   // UNICODE_TO_GBK[7258] := 16#5960;
   // UNICODE_TO_GBK[7259] := 16#B5EC;
   // UNICODE_TO_GBK[7260] := 16#5961;
   // UNICODE_TO_GBK[7261] := 16#8A53;
   // UNICODE_TO_GBK[7262] := 16#5962;
   // UNICODE_TO_GBK[7263] := 16#C9DD;
   // UNICODE_TO_GBK[7264] := 16#5963;
   // UNICODE_TO_GBK[7265] := 16#8A54;
   // UNICODE_TO_GBK[7266] := 16#5964;
   // UNICODE_TO_GBK[7267] := 16#8A55;
   // UNICODE_TO_GBK[7268] := 16#5965;
   // UNICODE_TO_GBK[7269] := 16#B0C2;
   // UNICODE_TO_GBK[7270] := 16#5966;
   // UNICODE_TO_GBK[7271] := 16#8A56;
   // UNICODE_TO_GBK[7272] := 16#5967;
   // UNICODE_TO_GBK[7273] := 16#8A57;
   // UNICODE_TO_GBK[7274] := 16#5968;
   // UNICODE_TO_GBK[7275] := 16#8A58;
   // UNICODE_TO_GBK[7276] := 16#5969;
   // UNICODE_TO_GBK[7277] := 16#8A59;
   // UNICODE_TO_GBK[7278] := 16#596A;
   // UNICODE_TO_GBK[7279] := 16#8A5A;
   // UNICODE_TO_GBK[7280] := 16#596B;
   // UNICODE_TO_GBK[7281] := 16#8A5B;
   // UNICODE_TO_GBK[7282] := 16#596C;
   // UNICODE_TO_GBK[7283] := 16#8A5C;
   // UNICODE_TO_GBK[7284] := 16#596D;
   // UNICODE_TO_GBK[7285] := 16#8A5D;
   // UNICODE_TO_GBK[7286] := 16#596E;
   // UNICODE_TO_GBK[7287] := 16#8A5E;
   // UNICODE_TO_GBK[7288] := 16#596F;
   // UNICODE_TO_GBK[7289] := 16#8A5F;
   // UNICODE_TO_GBK[7290] := 16#5970;
   // UNICODE_TO_GBK[7291] := 16#8A60;
   // UNICODE_TO_GBK[7292] := 16#5971;
   // UNICODE_TO_GBK[7293] := 16#8A61;
   // UNICODE_TO_GBK[7294] := 16#5972;
   // UNICODE_TO_GBK[7295] := 16#8A62;
   // UNICODE_TO_GBK[7296] := 16#5973;
   // UNICODE_TO_GBK[7297] := 16#C5AE;
   // UNICODE_TO_GBK[7298] := 16#5974;
   // UNICODE_TO_GBK[7299] := 16#C5AB;
   // UNICODE_TO_GBK[7300] := 16#5975;
   // UNICODE_TO_GBK[7301] := 16#8A63;
   // UNICODE_TO_GBK[7302] := 16#5976;
   // UNICODE_TO_GBK[7303] := 16#C4CC;
   // UNICODE_TO_GBK[7304] := 16#5977;
   // UNICODE_TO_GBK[7305] := 16#8A64;
   // UNICODE_TO_GBK[7306] := 16#5978;
   // UNICODE_TO_GBK[7307] := 16#BCE9;
   // UNICODE_TO_GBK[7308] := 16#5979;
   // UNICODE_TO_GBK[7309] := 16#CBFD;
   // UNICODE_TO_GBK[7310] := 16#597A;
   // UNICODE_TO_GBK[7311] := 16#8A65;
   // UNICODE_TO_GBK[7312] := 16#597B;
   // UNICODE_TO_GBK[7313] := 16#8A66;
   // UNICODE_TO_GBK[7314] := 16#597C;
   // UNICODE_TO_GBK[7315] := 16#8A67;
   // UNICODE_TO_GBK[7316] := 16#597D;
   // UNICODE_TO_GBK[7317] := 16#BAC3;
   // UNICODE_TO_GBK[7318] := 16#597E;
   // UNICODE_TO_GBK[7319] := 16#8A68;
   // UNICODE_TO_GBK[7320] := 16#597F;
   // UNICODE_TO_GBK[7321] := 16#8A69;
   // UNICODE_TO_GBK[7322] := 16#5980;
   // UNICODE_TO_GBK[7323] := 16#8A6A;
   // UNICODE_TO_GBK[7324] := 16#5981;
   // UNICODE_TO_GBK[7325] := 16#E5F9;
   // UNICODE_TO_GBK[7326] := 16#5982;
   // UNICODE_TO_GBK[7327] := 16#C8E7;
   // UNICODE_TO_GBK[7328] := 16#5983;
   // UNICODE_TO_GBK[7329] := 16#E5FA;
   // UNICODE_TO_GBK[7330] := 16#5984;
   // UNICODE_TO_GBK[7331] := 16#CDFD;
   // UNICODE_TO_GBK[7332] := 16#5985;
   // UNICODE_TO_GBK[7333] := 16#8A6B;
   // UNICODE_TO_GBK[7334] := 16#5986;
   // UNICODE_TO_GBK[7335] := 16#D7B1;
   // UNICODE_TO_GBK[7336] := 16#5987;
   // UNICODE_TO_GBK[7337] := 16#B8BE;
   // UNICODE_TO_GBK[7338] := 16#5988;
   // UNICODE_TO_GBK[7339] := 16#C2E8;
   // UNICODE_TO_GBK[7340] := 16#5989;
   // UNICODE_TO_GBK[7341] := 16#8A6C;
   // UNICODE_TO_GBK[7342] := 16#598A;
   // UNICODE_TO_GBK[7343] := 16#C8D1;
   // UNICODE_TO_GBK[7344] := 16#598B;
   // UNICODE_TO_GBK[7345] := 16#8A6D;
   // UNICODE_TO_GBK[7346] := 16#598C;
   // UNICODE_TO_GBK[7347] := 16#8A6E;
   // UNICODE_TO_GBK[7348] := 16#598D;
   // UNICODE_TO_GBK[7349] := 16#E5FB;
   // UNICODE_TO_GBK[7350] := 16#598E;
   // UNICODE_TO_GBK[7351] := 16#8A6F;
   // UNICODE_TO_GBK[7352] := 16#598F;
   // UNICODE_TO_GBK[7353] := 16#8A70;
   // UNICODE_TO_GBK[7354] := 16#5990;
   // UNICODE_TO_GBK[7355] := 16#8A71;
   // UNICODE_TO_GBK[7356] := 16#5991;
   // UNICODE_TO_GBK[7357] := 16#8A72;
   // UNICODE_TO_GBK[7358] := 16#5992;
   // UNICODE_TO_GBK[7359] := 16#B6CA;
   // UNICODE_TO_GBK[7360] := 16#5993;
   // UNICODE_TO_GBK[7361] := 16#BCCB;
   // UNICODE_TO_GBK[7362] := 16#5994;
   // UNICODE_TO_GBK[7363] := 16#8A73;
   // UNICODE_TO_GBK[7364] := 16#5995;
   // UNICODE_TO_GBK[7365] := 16#8A74;
   // UNICODE_TO_GBK[7366] := 16#5996;
   // UNICODE_TO_GBK[7367] := 16#D1FD;
   // UNICODE_TO_GBK[7368] := 16#5997;
   // UNICODE_TO_GBK[7369] := 16#E6A1;
   // UNICODE_TO_GBK[7370] := 16#5998;
   // UNICODE_TO_GBK[7371] := 16#8A75;
   // UNICODE_TO_GBK[7372] := 16#5999;
   // UNICODE_TO_GBK[7373] := 16#C3EE;
   // UNICODE_TO_GBK[7374] := 16#599A;
   // UNICODE_TO_GBK[7375] := 16#8A76;
   // UNICODE_TO_GBK[7376] := 16#599B;
   // UNICODE_TO_GBK[7377] := 16#8A77;
   // UNICODE_TO_GBK[7378] := 16#599C;
   // UNICODE_TO_GBK[7379] := 16#8A78;
   // UNICODE_TO_GBK[7380] := 16#599D;
   // UNICODE_TO_GBK[7381] := 16#8A79;
   // UNICODE_TO_GBK[7382] := 16#599E;
   // UNICODE_TO_GBK[7383] := 16#E6A4;
   // UNICODE_TO_GBK[7384] := 16#599F;
   // UNICODE_TO_GBK[7385] := 16#8A7A;
   // UNICODE_TO_GBK[7386] := 16#59A0;
   // UNICODE_TO_GBK[7387] := 16#8A7B;
   // UNICODE_TO_GBK[7388] := 16#59A1;
   // UNICODE_TO_GBK[7389] := 16#8A7C;
   // UNICODE_TO_GBK[7390] := 16#59A2;
   // UNICODE_TO_GBK[7391] := 16#8A7D;
   // UNICODE_TO_GBK[7392] := 16#59A3;
   // UNICODE_TO_GBK[7393] := 16#E5FE;
   // UNICODE_TO_GBK[7394] := 16#59A4;
   // UNICODE_TO_GBK[7395] := 16#E6A5;
   // UNICODE_TO_GBK[7396] := 16#59A5;
   // UNICODE_TO_GBK[7397] := 16#CDD7;
   // UNICODE_TO_GBK[7398] := 16#59A6;
   // UNICODE_TO_GBK[7399] := 16#8A7E;
   // UNICODE_TO_GBK[7400] := 16#59A7;
   // UNICODE_TO_GBK[7401] := 16#8A80;
   // UNICODE_TO_GBK[7402] := 16#59A8;
   // UNICODE_TO_GBK[7403] := 16#B7C1;
   // UNICODE_TO_GBK[7404] := 16#59A9;
   // UNICODE_TO_GBK[7405] := 16#E5FC;
   // UNICODE_TO_GBK[7406] := 16#59AA;
   // UNICODE_TO_GBK[7407] := 16#E5FD;
   // UNICODE_TO_GBK[7408] := 16#59AB;
   // UNICODE_TO_GBK[7409] := 16#E6A3;
   // UNICODE_TO_GBK[7410] := 16#59AC;
   // UNICODE_TO_GBK[7411] := 16#8A81;
   // UNICODE_TO_GBK[7412] := 16#59AD;
   // UNICODE_TO_GBK[7413] := 16#8A82;
   // UNICODE_TO_GBK[7414] := 16#59AE;
   // UNICODE_TO_GBK[7415] := 16#C4DD;
   // UNICODE_TO_GBK[7416] := 16#59AF;
   // UNICODE_TO_GBK[7417] := 16#E6A8;
   // UNICODE_TO_GBK[7418] := 16#59B0;
   // UNICODE_TO_GBK[7419] := 16#8A83;
   // UNICODE_TO_GBK[7420] := 16#59B1;
   // UNICODE_TO_GBK[7421] := 16#8A84;
   // UNICODE_TO_GBK[7422] := 16#59B2;
   // UNICODE_TO_GBK[7423] := 16#E6A7;
   // UNICODE_TO_GBK[7424] := 16#59B3;
   // UNICODE_TO_GBK[7425] := 16#8A85;
   // UNICODE_TO_GBK[7426] := 16#59B4;
   // UNICODE_TO_GBK[7427] := 16#8A86;
   // UNICODE_TO_GBK[7428] := 16#59B5;
   // UNICODE_TO_GBK[7429] := 16#8A87;
   // UNICODE_TO_GBK[7430] := 16#59B6;
   // UNICODE_TO_GBK[7431] := 16#8A88;
   // UNICODE_TO_GBK[7432] := 16#59B7;
   // UNICODE_TO_GBK[7433] := 16#8A89;
   // UNICODE_TO_GBK[7434] := 16#59B8;
   // UNICODE_TO_GBK[7435] := 16#8A8A;
   // UNICODE_TO_GBK[7436] := 16#59B9;
   // UNICODE_TO_GBK[7437] := 16#C3C3;
   // UNICODE_TO_GBK[7438] := 16#59BA;
   // UNICODE_TO_GBK[7439] := 16#8A8B;
   // UNICODE_TO_GBK[7440] := 16#59BB;
   // UNICODE_TO_GBK[7441] := 16#C6DE;
   // UNICODE_TO_GBK[7442] := 16#59BC;
   // UNICODE_TO_GBK[7443] := 16#8A8C;
   // UNICODE_TO_GBK[7444] := 16#59BD;
   // UNICODE_TO_GBK[7445] := 16#8A8D;
   // UNICODE_TO_GBK[7446] := 16#59BE;
   // UNICODE_TO_GBK[7447] := 16#E6AA;
   // UNICODE_TO_GBK[7448] := 16#59BF;
   // UNICODE_TO_GBK[7449] := 16#8A8E;
   // UNICODE_TO_GBK[7450] := 16#59C0;
   // UNICODE_TO_GBK[7451] := 16#8A8F;
   // UNICODE_TO_GBK[7452] := 16#59C1;
   // UNICODE_TO_GBK[7453] := 16#8A90;
   // UNICODE_TO_GBK[7454] := 16#59C2;
   // UNICODE_TO_GBK[7455] := 16#8A91;
   // UNICODE_TO_GBK[7456] := 16#59C3;
   // UNICODE_TO_GBK[7457] := 16#8A92;
   // UNICODE_TO_GBK[7458] := 16#59C4;
   // UNICODE_TO_GBK[7459] := 16#8A93;
   // UNICODE_TO_GBK[7460] := 16#59C5;
   // UNICODE_TO_GBK[7461] := 16#8A94;
   // UNICODE_TO_GBK[7462] := 16#59C6;
   // UNICODE_TO_GBK[7463] := 16#C4B7;
   // UNICODE_TO_GBK[7464] := 16#59C7;
   // UNICODE_TO_GBK[7465] := 16#8A95;
   // UNICODE_TO_GBK[7466] := 16#59C8;
   // UNICODE_TO_GBK[7467] := 16#8A96;
   // UNICODE_TO_GBK[7468] := 16#59C9;
   // UNICODE_TO_GBK[7469] := 16#8A97;
   // UNICODE_TO_GBK[7470] := 16#59CA;
   // UNICODE_TO_GBK[7471] := 16#E6A2;
   // UNICODE_TO_GBK[7472] := 16#59CB;
   // UNICODE_TO_GBK[7473] := 16#CABC;
   // UNICODE_TO_GBK[7474] := 16#59CC;
   // UNICODE_TO_GBK[7475] := 16#8A98;
   // UNICODE_TO_GBK[7476] := 16#59CD;
   // UNICODE_TO_GBK[7477] := 16#8A99;
   // UNICODE_TO_GBK[7478] := 16#59CE;
   // UNICODE_TO_GBK[7479] := 16#8A9A;
   // UNICODE_TO_GBK[7480] := 16#59CF;
   // UNICODE_TO_GBK[7481] := 16#8A9B;
   // UNICODE_TO_GBK[7482] := 16#59D0;
   // UNICODE_TO_GBK[7483] := 16#BDE3;
   // UNICODE_TO_GBK[7484] := 16#59D1;
   // UNICODE_TO_GBK[7485] := 16#B9C3;
   // UNICODE_TO_GBK[7486] := 16#59D2;
   // UNICODE_TO_GBK[7487] := 16#E6A6;
   // UNICODE_TO_GBK[7488] := 16#59D3;
   // UNICODE_TO_GBK[7489] := 16#D0D5;
   // UNICODE_TO_GBK[7490] := 16#59D4;
   // UNICODE_TO_GBK[7491] := 16#CEAF;
   // UNICODE_TO_GBK[7492] := 16#59D5;
   // UNICODE_TO_GBK[7493] := 16#8A9C;
   // UNICODE_TO_GBK[7494] := 16#59D6;
   // UNICODE_TO_GBK[7495] := 16#8A9D;
   // UNICODE_TO_GBK[7496] := 16#59D7;
   // UNICODE_TO_GBK[7497] := 16#E6A9;
   // UNICODE_TO_GBK[7498] := 16#59D8;
   // UNICODE_TO_GBK[7499] := 16#E6B0;
   // UNICODE_TO_GBK[7500] := 16#59D9;
   // UNICODE_TO_GBK[7501] := 16#8A9E;
   // UNICODE_TO_GBK[7502] := 16#59DA;
   // UNICODE_TO_GBK[7503] := 16#D2A6;
   // UNICODE_TO_GBK[7504] := 16#59DB;
   // UNICODE_TO_GBK[7505] := 16#8A9F;
   // UNICODE_TO_GBK[7506] := 16#59DC;
   // UNICODE_TO_GBK[7507] := 16#BDAA;
   // UNICODE_TO_GBK[7508] := 16#59DD;
   // UNICODE_TO_GBK[7509] := 16#E6AD;
   // UNICODE_TO_GBK[7510] := 16#59DE;
   // UNICODE_TO_GBK[7511] := 16#8AA0;
   // UNICODE_TO_GBK[7512] := 16#59DF;
   // UNICODE_TO_GBK[7513] := 16#8AA1;
   // UNICODE_TO_GBK[7514] := 16#59E0;
   // UNICODE_TO_GBK[7515] := 16#8AA2;
   // UNICODE_TO_GBK[7516] := 16#59E1;
   // UNICODE_TO_GBK[7517] := 16#8AA3;
   // UNICODE_TO_GBK[7518] := 16#59E2;
   // UNICODE_TO_GBK[7519] := 16#8AA4;
   // UNICODE_TO_GBK[7520] := 16#59E3;
   // UNICODE_TO_GBK[7521] := 16#E6AF;
   // UNICODE_TO_GBK[7522] := 16#59E4;
   // UNICODE_TO_GBK[7523] := 16#8AA5;
   // UNICODE_TO_GBK[7524] := 16#59E5;
   // UNICODE_TO_GBK[7525] := 16#C0D1;
   // UNICODE_TO_GBK[7526] := 16#59E6;
   // UNICODE_TO_GBK[7527] := 16#8AA6;
   // UNICODE_TO_GBK[7528] := 16#59E7;
   // UNICODE_TO_GBK[7529] := 16#8AA7;
   // UNICODE_TO_GBK[7530] := 16#59E8;
   // UNICODE_TO_GBK[7531] := 16#D2CC;
   // UNICODE_TO_GBK[7532] := 16#59E9;
   // UNICODE_TO_GBK[7533] := 16#8AA8;
   // UNICODE_TO_GBK[7534] := 16#59EA;
   // UNICODE_TO_GBK[7535] := 16#8AA9;
   // UNICODE_TO_GBK[7536] := 16#59EB;
   // UNICODE_TO_GBK[7537] := 16#8AAA;
   // UNICODE_TO_GBK[7538] := 16#59EC;
   // UNICODE_TO_GBK[7539] := 16#BCA7;
   // UNICODE_TO_GBK[7540] := 16#59ED;
   // UNICODE_TO_GBK[7541] := 16#8AAB;
   // UNICODE_TO_GBK[7542] := 16#59EE;
   // UNICODE_TO_GBK[7543] := 16#8AAC;
   // UNICODE_TO_GBK[7544] := 16#59EF;
   // UNICODE_TO_GBK[7545] := 16#8AAD;
   // UNICODE_TO_GBK[7546] := 16#59F0;
   // UNICODE_TO_GBK[7547] := 16#8AAE;
   // UNICODE_TO_GBK[7548] := 16#59F1;
   // UNICODE_TO_GBK[7549] := 16#8AAF;
   // UNICODE_TO_GBK[7550] := 16#59F2;
   // UNICODE_TO_GBK[7551] := 16#8AB0;
   // UNICODE_TO_GBK[7552] := 16#59F3;
   // UNICODE_TO_GBK[7553] := 16#8AB1;
   // UNICODE_TO_GBK[7554] := 16#59F4;
   // UNICODE_TO_GBK[7555] := 16#8AB2;
   // UNICODE_TO_GBK[7556] := 16#59F5;
   // UNICODE_TO_GBK[7557] := 16#8AB3;
   // UNICODE_TO_GBK[7558] := 16#59F6;
   // UNICODE_TO_GBK[7559] := 16#8AB4;
   // UNICODE_TO_GBK[7560] := 16#59F7;
   // UNICODE_TO_GBK[7561] := 16#8AB5;
   // UNICODE_TO_GBK[7562] := 16#59F8;
   // UNICODE_TO_GBK[7563] := 16#8AB6;
   // UNICODE_TO_GBK[7564] := 16#59F9;
   // UNICODE_TO_GBK[7565] := 16#E6B1;
   // UNICODE_TO_GBK[7566] := 16#59FA;
   // UNICODE_TO_GBK[7567] := 16#8AB7;
   // UNICODE_TO_GBK[7568] := 16#59FB;
   // UNICODE_TO_GBK[7569] := 16#D2F6;
   // UNICODE_TO_GBK[7570] := 16#59FC;
   // UNICODE_TO_GBK[7571] := 16#8AB8;
   // UNICODE_TO_GBK[7572] := 16#59FD;
   // UNICODE_TO_GBK[7573] := 16#8AB9;
   // UNICODE_TO_GBK[7574] := 16#59FE;
   // UNICODE_TO_GBK[7575] := 16#8ABA;
   // UNICODE_TO_GBK[7576] := 16#59FF;
   // UNICODE_TO_GBK[7577] := 16#D7CB;
   // UNICODE_TO_GBK[7578] := 16#5A00;
   // UNICODE_TO_GBK[7579] := 16#8ABB;
   // UNICODE_TO_GBK[7580] := 16#5A01;
   // UNICODE_TO_GBK[7581] := 16#CDFE;
   // UNICODE_TO_GBK[7582] := 16#5A02;
   // UNICODE_TO_GBK[7583] := 16#8ABC;
   // UNICODE_TO_GBK[7584] := 16#5A03;
   // UNICODE_TO_GBK[7585] := 16#CDDE;
   // UNICODE_TO_GBK[7586] := 16#5A04;
   // UNICODE_TO_GBK[7587] := 16#C2A6;
   // UNICODE_TO_GBK[7588] := 16#5A05;
   // UNICODE_TO_GBK[7589] := 16#E6AB;
   // UNICODE_TO_GBK[7590] := 16#5A06;
   // UNICODE_TO_GBK[7591] := 16#E6AC;
   // UNICODE_TO_GBK[7592] := 16#5A07;
   // UNICODE_TO_GBK[7593] := 16#BDBF;
   // UNICODE_TO_GBK[7594] := 16#5A08;
   // UNICODE_TO_GBK[7595] := 16#E6AE;
   // UNICODE_TO_GBK[7596] := 16#5A09;
   // UNICODE_TO_GBK[7597] := 16#E6B3;
   // UNICODE_TO_GBK[7598] := 16#5A0A;
   // UNICODE_TO_GBK[7599] := 16#8ABD;
   // UNICODE_TO_GBK[7600] := 16#5A0B;
   // UNICODE_TO_GBK[7601] := 16#8ABE;
   // UNICODE_TO_GBK[7602] := 16#5A0C;
   // UNICODE_TO_GBK[7603] := 16#E6B2;
   // UNICODE_TO_GBK[7604] := 16#5A0D;
   // UNICODE_TO_GBK[7605] := 16#8ABF;
   // UNICODE_TO_GBK[7606] := 16#5A0E;
   // UNICODE_TO_GBK[7607] := 16#8AC0;
   // UNICODE_TO_GBK[7608] := 16#5A0F;
   // UNICODE_TO_GBK[7609] := 16#8AC1;
   // UNICODE_TO_GBK[7610] := 16#5A10;
   // UNICODE_TO_GBK[7611] := 16#8AC2;
   // UNICODE_TO_GBK[7612] := 16#5A11;
   // UNICODE_TO_GBK[7613] := 16#E6B6;
   // UNICODE_TO_GBK[7614] := 16#5A12;
   // UNICODE_TO_GBK[7615] := 16#8AC3;
   // UNICODE_TO_GBK[7616] := 16#5A13;
   // UNICODE_TO_GBK[7617] := 16#E6B8;
   // UNICODE_TO_GBK[7618] := 16#5A14;
   // UNICODE_TO_GBK[7619] := 16#8AC4;
   // UNICODE_TO_GBK[7620] := 16#5A15;
   // UNICODE_TO_GBK[7621] := 16#8AC5;
   // UNICODE_TO_GBK[7622] := 16#5A16;
   // UNICODE_TO_GBK[7623] := 16#8AC6;
   // UNICODE_TO_GBK[7624] := 16#5A17;
   // UNICODE_TO_GBK[7625] := 16#8AC7;
   // UNICODE_TO_GBK[7626] := 16#5A18;
   // UNICODE_TO_GBK[7627] := 16#C4EF;
   // UNICODE_TO_GBK[7628] := 16#5A19;
   // UNICODE_TO_GBK[7629] := 16#8AC8;
   // UNICODE_TO_GBK[7630] := 16#5A1A;
   // UNICODE_TO_GBK[7631] := 16#8AC9;
   // UNICODE_TO_GBK[7632] := 16#5A1B;
   // UNICODE_TO_GBK[7633] := 16#8ACA;
   // UNICODE_TO_GBK[7634] := 16#5A1C;
   // UNICODE_TO_GBK[7635] := 16#C4C8;
   // UNICODE_TO_GBK[7636] := 16#5A1D;
   // UNICODE_TO_GBK[7637] := 16#8ACB;
   // UNICODE_TO_GBK[7638] := 16#5A1E;
   // UNICODE_TO_GBK[7639] := 16#8ACC;
   // UNICODE_TO_GBK[7640] := 16#5A1F;
   // UNICODE_TO_GBK[7641] := 16#BEEA;
   // UNICODE_TO_GBK[7642] := 16#5A20;
   // UNICODE_TO_GBK[7643] := 16#C9EF;
   // UNICODE_TO_GBK[7644] := 16#5A21;
   // UNICODE_TO_GBK[7645] := 16#8ACD;
   // UNICODE_TO_GBK[7646] := 16#5A22;
   // UNICODE_TO_GBK[7647] := 16#8ACE;
   // UNICODE_TO_GBK[7648] := 16#5A23;
   // UNICODE_TO_GBK[7649] := 16#E6B7;
   // UNICODE_TO_GBK[7650] := 16#5A24;
   // UNICODE_TO_GBK[7651] := 16#8ACF;
   // UNICODE_TO_GBK[7652] := 16#5A25;
   // UNICODE_TO_GBK[7653] := 16#B6F0;
   // UNICODE_TO_GBK[7654] := 16#5A26;
   // UNICODE_TO_GBK[7655] := 16#8AD0;
   // UNICODE_TO_GBK[7656] := 16#5A27;
   // UNICODE_TO_GBK[7657] := 16#8AD1;
   // UNICODE_TO_GBK[7658] := 16#5A28;
   // UNICODE_TO_GBK[7659] := 16#8AD2;
   // UNICODE_TO_GBK[7660] := 16#5A29;
   // UNICODE_TO_GBK[7661] := 16#C3E4;
   // UNICODE_TO_GBK[7662] := 16#5A2A;
   // UNICODE_TO_GBK[7663] := 16#8AD3;
   // UNICODE_TO_GBK[7664] := 16#5A2B;
   // UNICODE_TO_GBK[7665] := 16#8AD4;
   // UNICODE_TO_GBK[7666] := 16#5A2C;
   // UNICODE_TO_GBK[7667] := 16#8AD5;
   // UNICODE_TO_GBK[7668] := 16#5A2D;
   // UNICODE_TO_GBK[7669] := 16#8AD6;
   // UNICODE_TO_GBK[7670] := 16#5A2E;
   // UNICODE_TO_GBK[7671] := 16#8AD7;
   // UNICODE_TO_GBK[7672] := 16#5A2F;
   // UNICODE_TO_GBK[7673] := 16#8AD8;
   // UNICODE_TO_GBK[7674] := 16#5A30;
   // UNICODE_TO_GBK[7675] := 16#8AD9;
   // UNICODE_TO_GBK[7676] := 16#5A31;
   // UNICODE_TO_GBK[7677] := 16#D3E9;
   // UNICODE_TO_GBK[7678] := 16#5A32;
   // UNICODE_TO_GBK[7679] := 16#E6B4;
   // UNICODE_TO_GBK[7680] := 16#5A33;
   // UNICODE_TO_GBK[7681] := 16#8ADA;
   // UNICODE_TO_GBK[7682] := 16#5A34;
   // UNICODE_TO_GBK[7683] := 16#E6B5;
   // UNICODE_TO_GBK[7684] := 16#5A35;
   // UNICODE_TO_GBK[7685] := 16#8ADB;
   // UNICODE_TO_GBK[7686] := 16#5A36;
   // UNICODE_TO_GBK[7687] := 16#C8A2;
   // UNICODE_TO_GBK[7688] := 16#5A37;
   // UNICODE_TO_GBK[7689] := 16#8ADC;
   // UNICODE_TO_GBK[7690] := 16#5A38;
   // UNICODE_TO_GBK[7691] := 16#8ADD;
   // UNICODE_TO_GBK[7692] := 16#5A39;
   // UNICODE_TO_GBK[7693] := 16#8ADE;
   // UNICODE_TO_GBK[7694] := 16#5A3A;
   // UNICODE_TO_GBK[7695] := 16#8ADF;
   // UNICODE_TO_GBK[7696] := 16#5A3B;
   // UNICODE_TO_GBK[7697] := 16#8AE0;
   // UNICODE_TO_GBK[7698] := 16#5A3C;
   // UNICODE_TO_GBK[7699] := 16#E6BD;
   // UNICODE_TO_GBK[7700] := 16#5A3D;
   // UNICODE_TO_GBK[7701] := 16#8AE1;
   // UNICODE_TO_GBK[7702] := 16#5A3E;
   // UNICODE_TO_GBK[7703] := 16#8AE2;
   // UNICODE_TO_GBK[7704] := 16#5A3F;
   // UNICODE_TO_GBK[7705] := 16#8AE3;
   // UNICODE_TO_GBK[7706] := 16#5A40;
   // UNICODE_TO_GBK[7707] := 16#E6B9;
   // UNICODE_TO_GBK[7708] := 16#5A41;
   // UNICODE_TO_GBK[7709] := 16#8AE4;
   // UNICODE_TO_GBK[7710] := 16#5A42;
   // UNICODE_TO_GBK[7711] := 16#8AE5;
   // UNICODE_TO_GBK[7712] := 16#5A43;
   // UNICODE_TO_GBK[7713] := 16#8AE6;
   // UNICODE_TO_GBK[7714] := 16#5A44;
   // UNICODE_TO_GBK[7715] := 16#8AE7;
   // UNICODE_TO_GBK[7716] := 16#5A45;
   // UNICODE_TO_GBK[7717] := 16#8AE8;
   // UNICODE_TO_GBK[7718] := 16#5A46;
   // UNICODE_TO_GBK[7719] := 16#C6C5;
   // UNICODE_TO_GBK[7720] := 16#5A47;
   // UNICODE_TO_GBK[7721] := 16#8AE9;
   // UNICODE_TO_GBK[7722] := 16#5A48;
   // UNICODE_TO_GBK[7723] := 16#8AEA;
   // UNICODE_TO_GBK[7724] := 16#5A49;
   // UNICODE_TO_GBK[7725] := 16#CDF1;
   // UNICODE_TO_GBK[7726] := 16#5A4A;
   // UNICODE_TO_GBK[7727] := 16#E6BB;
   // UNICODE_TO_GBK[7728] := 16#5A4B;
   // UNICODE_TO_GBK[7729] := 16#8AEB;
   // UNICODE_TO_GBK[7730] := 16#5A4C;
   // UNICODE_TO_GBK[7731] := 16#8AEC;
   // UNICODE_TO_GBK[7732] := 16#5A4D;
   // UNICODE_TO_GBK[7733] := 16#8AED;
   // UNICODE_TO_GBK[7734] := 16#5A4E;
   // UNICODE_TO_GBK[7735] := 16#8AEE;
   // UNICODE_TO_GBK[7736] := 16#5A4F;
   // UNICODE_TO_GBK[7737] := 16#8AEF;
   // UNICODE_TO_GBK[7738] := 16#5A50;
   // UNICODE_TO_GBK[7739] := 16#8AF0;
   // UNICODE_TO_GBK[7740] := 16#5A51;
   // UNICODE_TO_GBK[7741] := 16#8AF1;
   // UNICODE_TO_GBK[7742] := 16#5A52;
   // UNICODE_TO_GBK[7743] := 16#8AF2;
   // UNICODE_TO_GBK[7744] := 16#5A53;
   // UNICODE_TO_GBK[7745] := 16#8AF3;
   // UNICODE_TO_GBK[7746] := 16#5A54;
   // UNICODE_TO_GBK[7747] := 16#8AF4;
   // UNICODE_TO_GBK[7748] := 16#5A55;
   // UNICODE_TO_GBK[7749] := 16#E6BC;
   // UNICODE_TO_GBK[7750] := 16#5A56;
   // UNICODE_TO_GBK[7751] := 16#8AF5;
   // UNICODE_TO_GBK[7752] := 16#5A57;
   // UNICODE_TO_GBK[7753] := 16#8AF6;
   // UNICODE_TO_GBK[7754] := 16#5A58;
   // UNICODE_TO_GBK[7755] := 16#8AF7;
   // UNICODE_TO_GBK[7756] := 16#5A59;
   // UNICODE_TO_GBK[7757] := 16#8AF8;
   // UNICODE_TO_GBK[7758] := 16#5A5A;
   // UNICODE_TO_GBK[7759] := 16#BBE9;
   // UNICODE_TO_GBK[7760] := 16#5A5B;
   // UNICODE_TO_GBK[7761] := 16#8AF9;
   // UNICODE_TO_GBK[7762] := 16#5A5C;
   // UNICODE_TO_GBK[7763] := 16#8AFA;
   // UNICODE_TO_GBK[7764] := 16#5A5D;
   // UNICODE_TO_GBK[7765] := 16#8AFB;
   // UNICODE_TO_GBK[7766] := 16#5A5E;
   // UNICODE_TO_GBK[7767] := 16#8AFC;
   // UNICODE_TO_GBK[7768] := 16#5A5F;
   // UNICODE_TO_GBK[7769] := 16#8AFD;
   // UNICODE_TO_GBK[7770] := 16#5A60;
   // UNICODE_TO_GBK[7771] := 16#8AFE;
   // UNICODE_TO_GBK[7772] := 16#5A61;
   // UNICODE_TO_GBK[7773] := 16#8B40;
   // UNICODE_TO_GBK[7774] := 16#5A62;
   // UNICODE_TO_GBK[7775] := 16#E6BE;
   // UNICODE_TO_GBK[7776] := 16#5A63;
   // UNICODE_TO_GBK[7777] := 16#8B41;
   // UNICODE_TO_GBK[7778] := 16#5A64;
   // UNICODE_TO_GBK[7779] := 16#8B42;
   // UNICODE_TO_GBK[7780] := 16#5A65;
   // UNICODE_TO_GBK[7781] := 16#8B43;
   // UNICODE_TO_GBK[7782] := 16#5A66;
   // UNICODE_TO_GBK[7783] := 16#8B44;
   // UNICODE_TO_GBK[7784] := 16#5A67;
   // UNICODE_TO_GBK[7785] := 16#E6BA;
   // UNICODE_TO_GBK[7786] := 16#5A68;
   // UNICODE_TO_GBK[7787] := 16#8B45;
   // UNICODE_TO_GBK[7788] := 16#5A69;
   // UNICODE_TO_GBK[7789] := 16#8B46;
   // UNICODE_TO_GBK[7790] := 16#5A6A;
   // UNICODE_TO_GBK[7791] := 16#C0B7;
   // UNICODE_TO_GBK[7792] := 16#5A6B;
   // UNICODE_TO_GBK[7793] := 16#8B47;
   // UNICODE_TO_GBK[7794] := 16#5A6C;
   // UNICODE_TO_GBK[7795] := 16#8B48;
   // UNICODE_TO_GBK[7796] := 16#5A6D;
   // UNICODE_TO_GBK[7797] := 16#8B49;
   // UNICODE_TO_GBK[7798] := 16#5A6E;
   // UNICODE_TO_GBK[7799] := 16#8B4A;
   // UNICODE_TO_GBK[7800] := 16#5A6F;
   // UNICODE_TO_GBK[7801] := 16#8B4B;
   // UNICODE_TO_GBK[7802] := 16#5A70;
   // UNICODE_TO_GBK[7803] := 16#8B4C;
   // UNICODE_TO_GBK[7804] := 16#5A71;
   // UNICODE_TO_GBK[7805] := 16#8B4D;
   // UNICODE_TO_GBK[7806] := 16#5A72;
   // UNICODE_TO_GBK[7807] := 16#8B4E;
   // UNICODE_TO_GBK[7808] := 16#5A73;
   // UNICODE_TO_GBK[7809] := 16#8B4F;
   // UNICODE_TO_GBK[7810] := 16#5A74;
   // UNICODE_TO_GBK[7811] := 16#D3A4;
   // UNICODE_TO_GBK[7812] := 16#5A75;
   // UNICODE_TO_GBK[7813] := 16#E6BF;
   // UNICODE_TO_GBK[7814] := 16#5A76;
   // UNICODE_TO_GBK[7815] := 16#C9F4;
   // UNICODE_TO_GBK[7816] := 16#5A77;
   // UNICODE_TO_GBK[7817] := 16#E6C3;
   // UNICODE_TO_GBK[7818] := 16#5A78;
   // UNICODE_TO_GBK[7819] := 16#8B50;
   // UNICODE_TO_GBK[7820] := 16#5A79;
   // UNICODE_TO_GBK[7821] := 16#8B51;
   // UNICODE_TO_GBK[7822] := 16#5A7A;
   // UNICODE_TO_GBK[7823] := 16#E6C4;
   // UNICODE_TO_GBK[7824] := 16#5A7B;
   // UNICODE_TO_GBK[7825] := 16#8B52;
   // UNICODE_TO_GBK[7826] := 16#5A7C;
   // UNICODE_TO_GBK[7827] := 16#8B53;
   // UNICODE_TO_GBK[7828] := 16#5A7D;
   // UNICODE_TO_GBK[7829] := 16#8B54;
   // UNICODE_TO_GBK[7830] := 16#5A7E;
   // UNICODE_TO_GBK[7831] := 16#8B55;
   // UNICODE_TO_GBK[7832] := 16#5A7F;
   // UNICODE_TO_GBK[7833] := 16#D0F6;
   // UNICODE_TO_GBK[7834] := 16#5A80;
   // UNICODE_TO_GBK[7835] := 16#8B56;
   // UNICODE_TO_GBK[7836] := 16#5A81;
   // UNICODE_TO_GBK[7837] := 16#8B57;
   // UNICODE_TO_GBK[7838] := 16#5A82;
   // UNICODE_TO_GBK[7839] := 16#8B58;
   // UNICODE_TO_GBK[7840] := 16#5A83;
   // UNICODE_TO_GBK[7841] := 16#8B59;
   // UNICODE_TO_GBK[7842] := 16#5A84;
   // UNICODE_TO_GBK[7843] := 16#8B5A;
   // UNICODE_TO_GBK[7844] := 16#5A85;
   // UNICODE_TO_GBK[7845] := 16#8B5B;
   // UNICODE_TO_GBK[7846] := 16#5A86;
   // UNICODE_TO_GBK[7847] := 16#8B5C;
   // UNICODE_TO_GBK[7848] := 16#5A87;
   // UNICODE_TO_GBK[7849] := 16#8B5D;
   // UNICODE_TO_GBK[7850] := 16#5A88;
   // UNICODE_TO_GBK[7851] := 16#8B5E;
   // UNICODE_TO_GBK[7852] := 16#5A89;
   // UNICODE_TO_GBK[7853] := 16#8B5F;
   // UNICODE_TO_GBK[7854] := 16#5A8A;
   // UNICODE_TO_GBK[7855] := 16#8B60;
   // UNICODE_TO_GBK[7856] := 16#5A8B;
   // UNICODE_TO_GBK[7857] := 16#8B61;
   // UNICODE_TO_GBK[7858] := 16#5A8C;
   // UNICODE_TO_GBK[7859] := 16#8B62;
   // UNICODE_TO_GBK[7860] := 16#5A8D;
   // UNICODE_TO_GBK[7861] := 16#8B63;
   // UNICODE_TO_GBK[7862] := 16#5A8E;
   // UNICODE_TO_GBK[7863] := 16#8B64;
   // UNICODE_TO_GBK[7864] := 16#5A8F;
   // UNICODE_TO_GBK[7865] := 16#8B65;
   // UNICODE_TO_GBK[7866] := 16#5A90;
   // UNICODE_TO_GBK[7867] := 16#8B66;
   // UNICODE_TO_GBK[7868] := 16#5A91;
   // UNICODE_TO_GBK[7869] := 16#8B67;
   // UNICODE_TO_GBK[7870] := 16#5A92;
   // UNICODE_TO_GBK[7871] := 16#C3BD;
   // UNICODE_TO_GBK[7872] := 16#5A93;
   // UNICODE_TO_GBK[7873] := 16#8B68;
   // UNICODE_TO_GBK[7874] := 16#5A94;
   // UNICODE_TO_GBK[7875] := 16#8B69;
   // UNICODE_TO_GBK[7876] := 16#5A95;
   // UNICODE_TO_GBK[7877] := 16#8B6A;
   // UNICODE_TO_GBK[7878] := 16#5A96;
   // UNICODE_TO_GBK[7879] := 16#8B6B;
   // UNICODE_TO_GBK[7880] := 16#5A97;
   // UNICODE_TO_GBK[7881] := 16#8B6C;
   // UNICODE_TO_GBK[7882] := 16#5A98;
   // UNICODE_TO_GBK[7883] := 16#8B6D;
   // UNICODE_TO_GBK[7884] := 16#5A99;
   // UNICODE_TO_GBK[7885] := 16#8B6E;
   // UNICODE_TO_GBK[7886] := 16#5A9A;
   // UNICODE_TO_GBK[7887] := 16#C3C4;
   // UNICODE_TO_GBK[7888] := 16#5A9B;
   // UNICODE_TO_GBK[7889] := 16#E6C2;
   // UNICODE_TO_GBK[7890] := 16#5A9C;
   // UNICODE_TO_GBK[7891] := 16#8B6F;
   // UNICODE_TO_GBK[7892] := 16#5A9D;
   // UNICODE_TO_GBK[7893] := 16#8B70;
   // UNICODE_TO_GBK[7894] := 16#5A9E;
   // UNICODE_TO_GBK[7895] := 16#8B71;
   // UNICODE_TO_GBK[7896] := 16#5A9F;
   // UNICODE_TO_GBK[7897] := 16#8B72;
   // UNICODE_TO_GBK[7898] := 16#5AA0;
   // UNICODE_TO_GBK[7899] := 16#8B73;
   // UNICODE_TO_GBK[7900] := 16#5AA1;
   // UNICODE_TO_GBK[7901] := 16#8B74;
   // UNICODE_TO_GBK[7902] := 16#5AA2;
   // UNICODE_TO_GBK[7903] := 16#8B75;
   // UNICODE_TO_GBK[7904] := 16#5AA3;
   // UNICODE_TO_GBK[7905] := 16#8B76;
   // UNICODE_TO_GBK[7906] := 16#5AA4;
   // UNICODE_TO_GBK[7907] := 16#8B77;
   // UNICODE_TO_GBK[7908] := 16#5AA5;
   // UNICODE_TO_GBK[7909] := 16#8B78;
   // UNICODE_TO_GBK[7910] := 16#5AA6;
   // UNICODE_TO_GBK[7911] := 16#8B79;
   // UNICODE_TO_GBK[7912] := 16#5AA7;
   // UNICODE_TO_GBK[7913] := 16#8B7A;
   // UNICODE_TO_GBK[7914] := 16#5AA8;
   // UNICODE_TO_GBK[7915] := 16#8B7B;
   // UNICODE_TO_GBK[7916] := 16#5AA9;
   // UNICODE_TO_GBK[7917] := 16#8B7C;
   // UNICODE_TO_GBK[7918] := 16#5AAA;
   // UNICODE_TO_GBK[7919] := 16#E6C1;
   // UNICODE_TO_GBK[7920] := 16#5AAB;
   // UNICODE_TO_GBK[7921] := 16#8B7D;
   // UNICODE_TO_GBK[7922] := 16#5AAC;
   // UNICODE_TO_GBK[7923] := 16#8B7E;
   // UNICODE_TO_GBK[7924] := 16#5AAD;
   // UNICODE_TO_GBK[7925] := 16#8B80;
   // UNICODE_TO_GBK[7926] := 16#5AAE;
   // UNICODE_TO_GBK[7927] := 16#8B81;
   // UNICODE_TO_GBK[7928] := 16#5AAF;
   // UNICODE_TO_GBK[7929] := 16#8B82;
   // UNICODE_TO_GBK[7930] := 16#5AB0;
   // UNICODE_TO_GBK[7931] := 16#8B83;
   // UNICODE_TO_GBK[7932] := 16#5AB1;
   // UNICODE_TO_GBK[7933] := 16#8B84;
   // UNICODE_TO_GBK[7934] := 16#5AB2;
   // UNICODE_TO_GBK[7935] := 16#E6C7;
   // UNICODE_TO_GBK[7936] := 16#5AB3;
   // UNICODE_TO_GBK[7937] := 16#CFB1;
   // UNICODE_TO_GBK[7938] := 16#5AB4;
   // UNICODE_TO_GBK[7939] := 16#8B85;
   // UNICODE_TO_GBK[7940] := 16#5AB5;
   // UNICODE_TO_GBK[7941] := 16#EBF4;
   // UNICODE_TO_GBK[7942] := 16#5AB6;
   // UNICODE_TO_GBK[7943] := 16#8B86;
   // UNICODE_TO_GBK[7944] := 16#5AB7;
   // UNICODE_TO_GBK[7945] := 16#8B87;
   // UNICODE_TO_GBK[7946] := 16#5AB8;
   // UNICODE_TO_GBK[7947] := 16#E6CA;
   // UNICODE_TO_GBK[7948] := 16#5AB9;
   // UNICODE_TO_GBK[7949] := 16#8B88;
   // UNICODE_TO_GBK[7950] := 16#5ABA;
   // UNICODE_TO_GBK[7951] := 16#8B89;
   // UNICODE_TO_GBK[7952] := 16#5ABB;
   // UNICODE_TO_GBK[7953] := 16#8B8A;
   // UNICODE_TO_GBK[7954] := 16#5ABC;
   // UNICODE_TO_GBK[7955] := 16#8B8B;
   // UNICODE_TO_GBK[7956] := 16#5ABD;
   // UNICODE_TO_GBK[7957] := 16#8B8C;
   // UNICODE_TO_GBK[7958] := 16#5ABE;
   // UNICODE_TO_GBK[7959] := 16#E6C5;
   // UNICODE_TO_GBK[7960] := 16#5ABF;
   // UNICODE_TO_GBK[7961] := 16#8B8D;
   // UNICODE_TO_GBK[7962] := 16#5AC0;
   // UNICODE_TO_GBK[7963] := 16#8B8E;
   // UNICODE_TO_GBK[7964] := 16#5AC1;
   // UNICODE_TO_GBK[7965] := 16#BCDE;
   // UNICODE_TO_GBK[7966] := 16#5AC2;
   // UNICODE_TO_GBK[7967] := 16#C9A9;
   // UNICODE_TO_GBK[7968] := 16#5AC3;
   // UNICODE_TO_GBK[7969] := 16#8B8F;
   // UNICODE_TO_GBK[7970] := 16#5AC4;
   // UNICODE_TO_GBK[7971] := 16#8B90;
   // UNICODE_TO_GBK[7972] := 16#5AC5;
   // UNICODE_TO_GBK[7973] := 16#8B91;
   // UNICODE_TO_GBK[7974] := 16#5AC6;
   // UNICODE_TO_GBK[7975] := 16#8B92;
   // UNICODE_TO_GBK[7976] := 16#5AC7;
   // UNICODE_TO_GBK[7977] := 16#8B93;
   // UNICODE_TO_GBK[7978] := 16#5AC8;
   // UNICODE_TO_GBK[7979] := 16#8B94;
   // UNICODE_TO_GBK[7980] := 16#5AC9;
   // UNICODE_TO_GBK[7981] := 16#BCB5;
   // UNICODE_TO_GBK[7982] := 16#5ACA;
   // UNICODE_TO_GBK[7983] := 16#8B95;
   // UNICODE_TO_GBK[7984] := 16#5ACB;
   // UNICODE_TO_GBK[7985] := 16#8B96;
   // UNICODE_TO_GBK[7986] := 16#5ACC;
   // UNICODE_TO_GBK[7987] := 16#CFD3;
   // UNICODE_TO_GBK[7988] := 16#5ACD;
   // UNICODE_TO_GBK[7989] := 16#8B97;
   // UNICODE_TO_GBK[7990] := 16#5ACE;
   // UNICODE_TO_GBK[7991] := 16#8B98;
   // UNICODE_TO_GBK[7992] := 16#5ACF;
   // UNICODE_TO_GBK[7993] := 16#8B99;
   // UNICODE_TO_GBK[7994] := 16#5AD0;
   // UNICODE_TO_GBK[7995] := 16#8B9A;
   // UNICODE_TO_GBK[7996] := 16#5AD1;
   // UNICODE_TO_GBK[7997] := 16#8B9B;
   // UNICODE_TO_GBK[7998] := 16#5AD2;
   // UNICODE_TO_GBK[7999] := 16#E6C8;
   // UNICODE_TO_GBK[8000] := 16#5AD3;
   // UNICODE_TO_GBK[8001] := 16#8B9C;
   // UNICODE_TO_GBK[8002] := 16#5AD4;
   // UNICODE_TO_GBK[8003] := 16#E6C9;
   // UNICODE_TO_GBK[8004] := 16#5AD5;
   // UNICODE_TO_GBK[8005] := 16#8B9D;
   // UNICODE_TO_GBK[8006] := 16#5AD6;
   // UNICODE_TO_GBK[8007] := 16#E6CE;
   // UNICODE_TO_GBK[8008] := 16#5AD7;
   // UNICODE_TO_GBK[8009] := 16#8B9E;
   // UNICODE_TO_GBK[8010] := 16#5AD8;
   // UNICODE_TO_GBK[8011] := 16#E6D0;
   // UNICODE_TO_GBK[8012] := 16#5AD9;
   // UNICODE_TO_GBK[8013] := 16#8B9F;
   // UNICODE_TO_GBK[8014] := 16#5ADA;
   // UNICODE_TO_GBK[8015] := 16#8BA0;
   // UNICODE_TO_GBK[8016] := 16#5ADB;
   // UNICODE_TO_GBK[8017] := 16#8BA1;
   // UNICODE_TO_GBK[8018] := 16#5ADC;
   // UNICODE_TO_GBK[8019] := 16#E6D1;
   // UNICODE_TO_GBK[8020] := 16#5ADD;
   // UNICODE_TO_GBK[8021] := 16#8BA2;
   // UNICODE_TO_GBK[8022] := 16#5ADE;
   // UNICODE_TO_GBK[8023] := 16#8BA3;
   // UNICODE_TO_GBK[8024] := 16#5ADF;
   // UNICODE_TO_GBK[8025] := 16#8BA4;
   // UNICODE_TO_GBK[8026] := 16#5AE0;
   // UNICODE_TO_GBK[8027] := 16#E6CB;
   // UNICODE_TO_GBK[8028] := 16#5AE1;
   // UNICODE_TO_GBK[8029] := 16#B5D5;
   // UNICODE_TO_GBK[8030] := 16#5AE2;
   // UNICODE_TO_GBK[8031] := 16#8BA5;
   // UNICODE_TO_GBK[8032] := 16#5AE3;
   // UNICODE_TO_GBK[8033] := 16#E6CC;
   // UNICODE_TO_GBK[8034] := 16#5AE4;
   // UNICODE_TO_GBK[8035] := 16#8BA6;
   // UNICODE_TO_GBK[8036] := 16#5AE5;
   // UNICODE_TO_GBK[8037] := 16#8BA7;
   // UNICODE_TO_GBK[8038] := 16#5AE6;
   // UNICODE_TO_GBK[8039] := 16#E6CF;
   // UNICODE_TO_GBK[8040] := 16#5AE7;
   // UNICODE_TO_GBK[8041] := 16#8BA8;
   // UNICODE_TO_GBK[8042] := 16#5AE8;
   // UNICODE_TO_GBK[8043] := 16#8BA9;
   // UNICODE_TO_GBK[8044] := 16#5AE9;
   // UNICODE_TO_GBK[8045] := 16#C4DB;
   // UNICODE_TO_GBK[8046] := 16#5AEA;
   // UNICODE_TO_GBK[8047] := 16#8BAA;
   // UNICODE_TO_GBK[8048] := 16#5AEB;
   // UNICODE_TO_GBK[8049] := 16#E6C6;
   // UNICODE_TO_GBK[8050] := 16#5AEC;
   // UNICODE_TO_GBK[8051] := 16#8BAB;
   // UNICODE_TO_GBK[8052] := 16#5AED;
   // UNICODE_TO_GBK[8053] := 16#8BAC;
   // UNICODE_TO_GBK[8054] := 16#5AEE;
   // UNICODE_TO_GBK[8055] := 16#8BAD;
   // UNICODE_TO_GBK[8056] := 16#5AEF;
   // UNICODE_TO_GBK[8057] := 16#8BAE;
   // UNICODE_TO_GBK[8058] := 16#5AF0;
   // UNICODE_TO_GBK[8059] := 16#8BAF;
   // UNICODE_TO_GBK[8060] := 16#5AF1;
   // UNICODE_TO_GBK[8061] := 16#E6CD;
   // UNICODE_TO_GBK[8062] := 16#5AF2;
   // UNICODE_TO_GBK[8063] := 16#8BB0;
   // UNICODE_TO_GBK[8064] := 16#5AF3;
   // UNICODE_TO_GBK[8065] := 16#8BB1;
   // UNICODE_TO_GBK[8066] := 16#5AF4;
   // UNICODE_TO_GBK[8067] := 16#8BB2;
   // UNICODE_TO_GBK[8068] := 16#5AF5;
   // UNICODE_TO_GBK[8069] := 16#8BB3;
   // UNICODE_TO_GBK[8070] := 16#5AF6;
   // UNICODE_TO_GBK[8071] := 16#8BB4;
   // UNICODE_TO_GBK[8072] := 16#5AF7;
   // UNICODE_TO_GBK[8073] := 16#8BB5;
   // UNICODE_TO_GBK[8074] := 16#5AF8;
   // UNICODE_TO_GBK[8075] := 16#8BB6;
   // UNICODE_TO_GBK[8076] := 16#5AF9;
   // UNICODE_TO_GBK[8077] := 16#8BB7;
   // UNICODE_TO_GBK[8078] := 16#5AFA;
   // UNICODE_TO_GBK[8079] := 16#8BB8;
   // UNICODE_TO_GBK[8080] := 16#5AFB;
   // UNICODE_TO_GBK[8081] := 16#8BB9;
   // UNICODE_TO_GBK[8082] := 16#5AFC;
   // UNICODE_TO_GBK[8083] := 16#8BBA;
   // UNICODE_TO_GBK[8084] := 16#5AFD;
   // UNICODE_TO_GBK[8085] := 16#8BBB;
   // UNICODE_TO_GBK[8086] := 16#5AFE;
   // UNICODE_TO_GBK[8087] := 16#8BBC;
   // UNICODE_TO_GBK[8088] := 16#5AFF;
   // UNICODE_TO_GBK[8089] := 16#8BBD;
   // UNICODE_TO_GBK[8090] := 16#5B00;
   // UNICODE_TO_GBK[8091] := 16#8BBE;
   // UNICODE_TO_GBK[8092] := 16#5B01;
   // UNICODE_TO_GBK[8093] := 16#8BBF;
   // UNICODE_TO_GBK[8094] := 16#5B02;
   // UNICODE_TO_GBK[8095] := 16#8BC0;
   // UNICODE_TO_GBK[8096] := 16#5B03;
   // UNICODE_TO_GBK[8097] := 16#8BC1;
   // UNICODE_TO_GBK[8098] := 16#5B04;
   // UNICODE_TO_GBK[8099] := 16#8BC2;
   // UNICODE_TO_GBK[8100] := 16#5B05;
   // UNICODE_TO_GBK[8101] := 16#8BC3;
   // UNICODE_TO_GBK[8102] := 16#5B06;
   // UNICODE_TO_GBK[8103] := 16#8BC4;
   // UNICODE_TO_GBK[8104] := 16#5B07;
   // UNICODE_TO_GBK[8105] := 16#8BC5;
   // UNICODE_TO_GBK[8106] := 16#5B08;
   // UNICODE_TO_GBK[8107] := 16#8BC6;
   // UNICODE_TO_GBK[8108] := 16#5B09;
   // UNICODE_TO_GBK[8109] := 16#E6D2;
   // UNICODE_TO_GBK[8110] := 16#5B0A;
   // UNICODE_TO_GBK[8111] := 16#8BC7;
   // UNICODE_TO_GBK[8112] := 16#5B0B;
   // UNICODE_TO_GBK[8113] := 16#8BC8;
   // UNICODE_TO_GBK[8114] := 16#5B0C;
   // UNICODE_TO_GBK[8115] := 16#8BC9;
   // UNICODE_TO_GBK[8116] := 16#5B0D;
   // UNICODE_TO_GBK[8117] := 16#8BCA;
   // UNICODE_TO_GBK[8118] := 16#5B0E;
   // UNICODE_TO_GBK[8119] := 16#8BCB;
   // UNICODE_TO_GBK[8120] := 16#5B0F;
   // UNICODE_TO_GBK[8121] := 16#8BCC;
   // UNICODE_TO_GBK[8122] := 16#5B10;
   // UNICODE_TO_GBK[8123] := 16#8BCD;
   // UNICODE_TO_GBK[8124] := 16#5B11;
   // UNICODE_TO_GBK[8125] := 16#8BCE;
   // UNICODE_TO_GBK[8126] := 16#5B12;
   // UNICODE_TO_GBK[8127] := 16#8BCF;
   // UNICODE_TO_GBK[8128] := 16#5B13;
   // UNICODE_TO_GBK[8129] := 16#8BD0;
   // UNICODE_TO_GBK[8130] := 16#5B14;
   // UNICODE_TO_GBK[8131] := 16#8BD1;
   // UNICODE_TO_GBK[8132] := 16#5B15;
   // UNICODE_TO_GBK[8133] := 16#8BD2;
   // UNICODE_TO_GBK[8134] := 16#5B16;
   // UNICODE_TO_GBK[8135] := 16#E6D4;
   // UNICODE_TO_GBK[8136] := 16#5B17;
   // UNICODE_TO_GBK[8137] := 16#E6D3;
   // UNICODE_TO_GBK[8138] := 16#5B18;
   // UNICODE_TO_GBK[8139] := 16#8BD3;
   // UNICODE_TO_GBK[8140] := 16#5B19;
   // UNICODE_TO_GBK[8141] := 16#8BD4;
   // UNICODE_TO_GBK[8142] := 16#5B1A;
   // UNICODE_TO_GBK[8143] := 16#8BD5;
   // UNICODE_TO_GBK[8144] := 16#5B1B;
   // UNICODE_TO_GBK[8145] := 16#8BD6;
   // UNICODE_TO_GBK[8146] := 16#5B1C;
   // UNICODE_TO_GBK[8147] := 16#8BD7;
   // UNICODE_TO_GBK[8148] := 16#5B1D;
   // UNICODE_TO_GBK[8149] := 16#8BD8;
   // UNICODE_TO_GBK[8150] := 16#5B1E;
   // UNICODE_TO_GBK[8151] := 16#8BD9;
   // UNICODE_TO_GBK[8152] := 16#5B1F;
   // UNICODE_TO_GBK[8153] := 16#8BDA;
   // UNICODE_TO_GBK[8154] := 16#5B20;
   // UNICODE_TO_GBK[8155] := 16#8BDB;
   // UNICODE_TO_GBK[8156] := 16#5B21;
   // UNICODE_TO_GBK[8157] := 16#8BDC;
   // UNICODE_TO_GBK[8158] := 16#5B22;
   // UNICODE_TO_GBK[8159] := 16#8BDD;
   // UNICODE_TO_GBK[8160] := 16#5B23;
   // UNICODE_TO_GBK[8161] := 16#8BDE;
   // UNICODE_TO_GBK[8162] := 16#5B24;
   // UNICODE_TO_GBK[8163] := 16#8BDF;
   // UNICODE_TO_GBK[8164] := 16#5B25;
   // UNICODE_TO_GBK[8165] := 16#8BE0;
   // UNICODE_TO_GBK[8166] := 16#5B26;
   // UNICODE_TO_GBK[8167] := 16#8BE1;
   // UNICODE_TO_GBK[8168] := 16#5B27;
   // UNICODE_TO_GBK[8169] := 16#8BE2;
   // UNICODE_TO_GBK[8170] := 16#5B28;
   // UNICODE_TO_GBK[8171] := 16#8BE3;
   // UNICODE_TO_GBK[8172] := 16#5B29;
   // UNICODE_TO_GBK[8173] := 16#8BE4;
   // UNICODE_TO_GBK[8174] := 16#5B2A;
   // UNICODE_TO_GBK[8175] := 16#8BE5;
   // UNICODE_TO_GBK[8176] := 16#5B2B;
   // UNICODE_TO_GBK[8177] := 16#8BE6;
   // UNICODE_TO_GBK[8178] := 16#5B2C;
   // UNICODE_TO_GBK[8179] := 16#8BE7;
   // UNICODE_TO_GBK[8180] := 16#5B2D;
   // UNICODE_TO_GBK[8181] := 16#8BE8;
   // UNICODE_TO_GBK[8182] := 16#5B2E;
   // UNICODE_TO_GBK[8183] := 16#8BE9;
   // UNICODE_TO_GBK[8184] := 16#5B2F;
   // UNICODE_TO_GBK[8185] := 16#8BEA;
   // UNICODE_TO_GBK[8186] := 16#5B30;
   // UNICODE_TO_GBK[8187] := 16#8BEB;
   // UNICODE_TO_GBK[8188] := 16#5B31;
   // UNICODE_TO_GBK[8189] := 16#8BEC;
   // UNICODE_TO_GBK[8190] := 16#5B32;
   // UNICODE_TO_GBK[8191] := 16#E6D5;
   // UNICODE_TO_GBK[8192] := 16#5B33;
   // UNICODE_TO_GBK[8193] := 16#8BED;
   // UNICODE_TO_GBK[8194] := 16#5B34;
   // UNICODE_TO_GBK[8195] := 16#D9F8;
   // UNICODE_TO_GBK[8196] := 16#5B35;
   // UNICODE_TO_GBK[8197] := 16#8BEE;
   // UNICODE_TO_GBK[8198] := 16#5B36;
   // UNICODE_TO_GBK[8199] := 16#8BEF;
   // UNICODE_TO_GBK[8200] := 16#5B37;
   // UNICODE_TO_GBK[8201] := 16#E6D6;
   // UNICODE_TO_GBK[8202] := 16#5B38;
   // UNICODE_TO_GBK[8203] := 16#8BF0;
   // UNICODE_TO_GBK[8204] := 16#5B39;
   // UNICODE_TO_GBK[8205] := 16#8BF1;
   // UNICODE_TO_GBK[8206] := 16#5B3A;
   // UNICODE_TO_GBK[8207] := 16#8BF2;
   // UNICODE_TO_GBK[8208] := 16#5B3B;
   // UNICODE_TO_GBK[8209] := 16#8BF3;
   // UNICODE_TO_GBK[8210] := 16#5B3C;
   // UNICODE_TO_GBK[8211] := 16#8BF4;
   // UNICODE_TO_GBK[8212] := 16#5B3D;
   // UNICODE_TO_GBK[8213] := 16#8BF5;
   // UNICODE_TO_GBK[8214] := 16#5B3E;
   // UNICODE_TO_GBK[8215] := 16#8BF6;
   // UNICODE_TO_GBK[8216] := 16#5B3F;
   // UNICODE_TO_GBK[8217] := 16#8BF7;
   // UNICODE_TO_GBK[8218] := 16#5B40;
   // UNICODE_TO_GBK[8219] := 16#E6D7;
   // UNICODE_TO_GBK[8220] := 16#5B41;
   // UNICODE_TO_GBK[8221] := 16#8BF8;
   // UNICODE_TO_GBK[8222] := 16#5B42;
   // UNICODE_TO_GBK[8223] := 16#8BF9;
   // UNICODE_TO_GBK[8224] := 16#5B43;
   // UNICODE_TO_GBK[8225] := 16#8BFA;
   // UNICODE_TO_GBK[8226] := 16#5B44;
   // UNICODE_TO_GBK[8227] := 16#8BFB;
   // UNICODE_TO_GBK[8228] := 16#5B45;
   // UNICODE_TO_GBK[8229] := 16#8BFC;
   // UNICODE_TO_GBK[8230] := 16#5B46;
   // UNICODE_TO_GBK[8231] := 16#8BFD;
   // UNICODE_TO_GBK[8232] := 16#5B47;
   // UNICODE_TO_GBK[8233] := 16#8BFE;
   // UNICODE_TO_GBK[8234] := 16#5B48;
   // UNICODE_TO_GBK[8235] := 16#8C40;
   // UNICODE_TO_GBK[8236] := 16#5B49;
   // UNICODE_TO_GBK[8237] := 16#8C41;
   // UNICODE_TO_GBK[8238] := 16#5B4A;
   // UNICODE_TO_GBK[8239] := 16#8C42;
   // UNICODE_TO_GBK[8240] := 16#5B4B;
   // UNICODE_TO_GBK[8241] := 16#8C43;
   // UNICODE_TO_GBK[8242] := 16#5B4C;
   // UNICODE_TO_GBK[8243] := 16#8C44;
   // UNICODE_TO_GBK[8244] := 16#5B4D;
   // UNICODE_TO_GBK[8245] := 16#8C45;
   // UNICODE_TO_GBK[8246] := 16#5B4E;
   // UNICODE_TO_GBK[8247] := 16#8C46;
   // UNICODE_TO_GBK[8248] := 16#5B4F;
   // UNICODE_TO_GBK[8249] := 16#8C47;
   // UNICODE_TO_GBK[8250] := 16#5B50;
   // UNICODE_TO_GBK[8251] := 16#D7D3;
   // UNICODE_TO_GBK[8252] := 16#5B51;
   // UNICODE_TO_GBK[8253] := 16#E6DD;
   // UNICODE_TO_GBK[8254] := 16#5B52;
   // UNICODE_TO_GBK[8255] := 16#8C48;
   // UNICODE_TO_GBK[8256] := 16#5B53;
   // UNICODE_TO_GBK[8257] := 16#E6DE;
   // UNICODE_TO_GBK[8258] := 16#5B54;
   // UNICODE_TO_GBK[8259] := 16#BFD7;
   // UNICODE_TO_GBK[8260] := 16#5B55;
   // UNICODE_TO_GBK[8261] := 16#D4D0;
   // UNICODE_TO_GBK[8262] := 16#5B56;
   // UNICODE_TO_GBK[8263] := 16#8C49;
   // UNICODE_TO_GBK[8264] := 16#5B57;
   // UNICODE_TO_GBK[8265] := 16#D7D6;
   // UNICODE_TO_GBK[8266] := 16#5B58;
   // UNICODE_TO_GBK[8267] := 16#B4E6;
   // UNICODE_TO_GBK[8268] := 16#5B59;
   // UNICODE_TO_GBK[8269] := 16#CBEF;
   // UNICODE_TO_GBK[8270] := 16#5B5A;
   // UNICODE_TO_GBK[8271] := 16#E6DA;
   // UNICODE_TO_GBK[8272] := 16#5B5B;
   // UNICODE_TO_GBK[8273] := 16#D8C3;
   // UNICODE_TO_GBK[8274] := 16#5B5C;
   // UNICODE_TO_GBK[8275] := 16#D7CE;
   // UNICODE_TO_GBK[8276] := 16#5B5D;
   // UNICODE_TO_GBK[8277] := 16#D0A2;
   // UNICODE_TO_GBK[8278] := 16#5B5E;
   // UNICODE_TO_GBK[8279] := 16#8C4A;
   // UNICODE_TO_GBK[8280] := 16#5B5F;
   // UNICODE_TO_GBK[8281] := 16#C3CF;
   // UNICODE_TO_GBK[8282] := 16#5B60;
   // UNICODE_TO_GBK[8283] := 16#8C4B;
   // UNICODE_TO_GBK[8284] := 16#5B61;
   // UNICODE_TO_GBK[8285] := 16#8C4C;
   // UNICODE_TO_GBK[8286] := 16#5B62;
   // UNICODE_TO_GBK[8287] := 16#E6DF;
   // UNICODE_TO_GBK[8288] := 16#5B63;
   // UNICODE_TO_GBK[8289] := 16#BCBE;
   // UNICODE_TO_GBK[8290] := 16#5B64;
   // UNICODE_TO_GBK[8291] := 16#B9C2;
   // UNICODE_TO_GBK[8292] := 16#5B65;
   // UNICODE_TO_GBK[8293] := 16#E6DB;
   // UNICODE_TO_GBK[8294] := 16#5B66;
   // UNICODE_TO_GBK[8295] := 16#D1A7;
   // UNICODE_TO_GBK[8296] := 16#5B67;
   // UNICODE_TO_GBK[8297] := 16#8C4D;
   // UNICODE_TO_GBK[8298] := 16#5B68;
   // UNICODE_TO_GBK[8299] := 16#8C4E;
   // UNICODE_TO_GBK[8300] := 16#5B69;
   // UNICODE_TO_GBK[8301] := 16#BAA2;
   // UNICODE_TO_GBK[8302] := 16#5B6A;
   // UNICODE_TO_GBK[8303] := 16#C2CF;
   // UNICODE_TO_GBK[8304] := 16#5B6B;
   // UNICODE_TO_GBK[8305] := 16#8C4F;
   // UNICODE_TO_GBK[8306] := 16#5B6C;
   // UNICODE_TO_GBK[8307] := 16#D8AB;
   // UNICODE_TO_GBK[8308] := 16#5B6D;
   // UNICODE_TO_GBK[8309] := 16#8C50;
   // UNICODE_TO_GBK[8310] := 16#5B6E;
   // UNICODE_TO_GBK[8311] := 16#8C51;
   // UNICODE_TO_GBK[8312] := 16#5B6F;
   // UNICODE_TO_GBK[8313] := 16#8C52;
   // UNICODE_TO_GBK[8314] := 16#5B70;
   // UNICODE_TO_GBK[8315] := 16#CAEB;
   // UNICODE_TO_GBK[8316] := 16#5B71;
   // UNICODE_TO_GBK[8317] := 16#E5EE;
   // UNICODE_TO_GBK[8318] := 16#5B72;
   // UNICODE_TO_GBK[8319] := 16#8C53;
   // UNICODE_TO_GBK[8320] := 16#5B73;
   // UNICODE_TO_GBK[8321] := 16#E6DC;
   // UNICODE_TO_GBK[8322] := 16#5B74;
   // UNICODE_TO_GBK[8323] := 16#8C54;
   // UNICODE_TO_GBK[8324] := 16#5B75;
   // UNICODE_TO_GBK[8325] := 16#B7F5;
   // UNICODE_TO_GBK[8326] := 16#5B76;
   // UNICODE_TO_GBK[8327] := 16#8C55;
   // UNICODE_TO_GBK[8328] := 16#5B77;
   // UNICODE_TO_GBK[8329] := 16#8C56;
   // UNICODE_TO_GBK[8330] := 16#5B78;
   // UNICODE_TO_GBK[8331] := 16#8C57;
   // UNICODE_TO_GBK[8332] := 16#5B79;
   // UNICODE_TO_GBK[8333] := 16#8C58;
   // UNICODE_TO_GBK[8334] := 16#5B7A;
   // UNICODE_TO_GBK[8335] := 16#C8E6;
   // UNICODE_TO_GBK[8336] := 16#5B7B;
   // UNICODE_TO_GBK[8337] := 16#8C59;
   // UNICODE_TO_GBK[8338] := 16#5B7C;
   // UNICODE_TO_GBK[8339] := 16#8C5A;
   // UNICODE_TO_GBK[8340] := 16#5B7D;
   // UNICODE_TO_GBK[8341] := 16#C4F5;
   // UNICODE_TO_GBK[8342] := 16#5B7E;
   // UNICODE_TO_GBK[8343] := 16#8C5B;
   // UNICODE_TO_GBK[8344] := 16#5B7F;
   // UNICODE_TO_GBK[8345] := 16#8C5C;
   // UNICODE_TO_GBK[8346] := 16#5B80;
   // UNICODE_TO_GBK[8347] := 16#E5B2;
   // UNICODE_TO_GBK[8348] := 16#5B81;
   // UNICODE_TO_GBK[8349] := 16#C4FE;
   // UNICODE_TO_GBK[8350] := 16#5B82;
   // UNICODE_TO_GBK[8351] := 16#8C5D;
   // UNICODE_TO_GBK[8352] := 16#5B83;
   // UNICODE_TO_GBK[8353] := 16#CBFC;
   // UNICODE_TO_GBK[8354] := 16#5B84;
   // UNICODE_TO_GBK[8355] := 16#E5B3;
   // UNICODE_TO_GBK[8356] := 16#5B85;
   // UNICODE_TO_GBK[8357] := 16#D5AC;
   // UNICODE_TO_GBK[8358] := 16#5B86;
   // UNICODE_TO_GBK[8359] := 16#8C5E;
   // UNICODE_TO_GBK[8360] := 16#5B87;
   // UNICODE_TO_GBK[8361] := 16#D3EE;
   // UNICODE_TO_GBK[8362] := 16#5B88;
   // UNICODE_TO_GBK[8363] := 16#CAD8;
   // UNICODE_TO_GBK[8364] := 16#5B89;
   // UNICODE_TO_GBK[8365] := 16#B0B2;
   // UNICODE_TO_GBK[8366] := 16#5B8A;
   // UNICODE_TO_GBK[8367] := 16#8C5F;
   // UNICODE_TO_GBK[8368] := 16#5B8B;
   // UNICODE_TO_GBK[8369] := 16#CBCE;
   // UNICODE_TO_GBK[8370] := 16#5B8C;
   // UNICODE_TO_GBK[8371] := 16#CDEA;
   // UNICODE_TO_GBK[8372] := 16#5B8D;
   // UNICODE_TO_GBK[8373] := 16#8C60;
   // UNICODE_TO_GBK[8374] := 16#5B8E;
   // UNICODE_TO_GBK[8375] := 16#8C61;
   // UNICODE_TO_GBK[8376] := 16#5B8F;
   // UNICODE_TO_GBK[8377] := 16#BAEA;
   // UNICODE_TO_GBK[8378] := 16#5B90;
   // UNICODE_TO_GBK[8379] := 16#8C62;
   // UNICODE_TO_GBK[8380] := 16#5B91;
   // UNICODE_TO_GBK[8381] := 16#8C63;
   // UNICODE_TO_GBK[8382] := 16#5B92;
   // UNICODE_TO_GBK[8383] := 16#8C64;
   // UNICODE_TO_GBK[8384] := 16#5B93;
   // UNICODE_TO_GBK[8385] := 16#E5B5;
   // UNICODE_TO_GBK[8386] := 16#5B94;
   // UNICODE_TO_GBK[8387] := 16#8C65;
   // UNICODE_TO_GBK[8388] := 16#5B95;
   // UNICODE_TO_GBK[8389] := 16#E5B4;
   // UNICODE_TO_GBK[8390] := 16#5B96;
   // UNICODE_TO_GBK[8391] := 16#8C66;
   // UNICODE_TO_GBK[8392] := 16#5B97;
   // UNICODE_TO_GBK[8393] := 16#D7DA;
   // UNICODE_TO_GBK[8394] := 16#5B98;
   // UNICODE_TO_GBK[8395] := 16#B9D9;
   // UNICODE_TO_GBK[8396] := 16#5B99;
   // UNICODE_TO_GBK[8397] := 16#D6E6;
   // UNICODE_TO_GBK[8398] := 16#5B9A;
   // UNICODE_TO_GBK[8399] := 16#B6A8;
   // UNICODE_TO_GBK[8400] := 16#5B9B;
   // UNICODE_TO_GBK[8401] := 16#CDF0;
   // UNICODE_TO_GBK[8402] := 16#5B9C;
   // UNICODE_TO_GBK[8403] := 16#D2CB;
   // UNICODE_TO_GBK[8404] := 16#5B9D;
   // UNICODE_TO_GBK[8405] := 16#B1A6;
   // UNICODE_TO_GBK[8406] := 16#5B9E;
   // UNICODE_TO_GBK[8407] := 16#CAB5;
   // UNICODE_TO_GBK[8408] := 16#5B9F;
   // UNICODE_TO_GBK[8409] := 16#8C67;
   // UNICODE_TO_GBK[8410] := 16#5BA0;
   // UNICODE_TO_GBK[8411] := 16#B3E8;
   // UNICODE_TO_GBK[8412] := 16#5BA1;
   // UNICODE_TO_GBK[8413] := 16#C9F3;
   // UNICODE_TO_GBK[8414] := 16#5BA2;
   // UNICODE_TO_GBK[8415] := 16#BFCD;
   // UNICODE_TO_GBK[8416] := 16#5BA3;
   // UNICODE_TO_GBK[8417] := 16#D0FB;
   // UNICODE_TO_GBK[8418] := 16#5BA4;
   // UNICODE_TO_GBK[8419] := 16#CAD2;
   // UNICODE_TO_GBK[8420] := 16#5BA5;
   // UNICODE_TO_GBK[8421] := 16#E5B6;
   // UNICODE_TO_GBK[8422] := 16#5BA6;
   // UNICODE_TO_GBK[8423] := 16#BBC2;
   // UNICODE_TO_GBK[8424] := 16#5BA7;
   // UNICODE_TO_GBK[8425] := 16#8C68;
   // UNICODE_TO_GBK[8426] := 16#5BA8;
   // UNICODE_TO_GBK[8427] := 16#8C69;
   // UNICODE_TO_GBK[8428] := 16#5BA9;
   // UNICODE_TO_GBK[8429] := 16#8C6A;
   // UNICODE_TO_GBK[8430] := 16#5BAA;
   // UNICODE_TO_GBK[8431] := 16#CFDC;
   // UNICODE_TO_GBK[8432] := 16#5BAB;
   // UNICODE_TO_GBK[8433] := 16#B9AC;
   // UNICODE_TO_GBK[8434] := 16#5BAC;
   // UNICODE_TO_GBK[8435] := 16#8C6B;
   // UNICODE_TO_GBK[8436] := 16#5BAD;
   // UNICODE_TO_GBK[8437] := 16#8C6C;
   // UNICODE_TO_GBK[8438] := 16#5BAE;
   // UNICODE_TO_GBK[8439] := 16#8C6D;
   // UNICODE_TO_GBK[8440] := 16#5BAF;
   // UNICODE_TO_GBK[8441] := 16#8C6E;
   // UNICODE_TO_GBK[8442] := 16#5BB0;
   // UNICODE_TO_GBK[8443] := 16#D4D7;
   // UNICODE_TO_GBK[8444] := 16#5BB1;
   // UNICODE_TO_GBK[8445] := 16#8C6F;
   // UNICODE_TO_GBK[8446] := 16#5BB2;
   // UNICODE_TO_GBK[8447] := 16#8C70;
   // UNICODE_TO_GBK[8448] := 16#5BB3;
   // UNICODE_TO_GBK[8449] := 16#BAA6;
   // UNICODE_TO_GBK[8450] := 16#5BB4;
   // UNICODE_TO_GBK[8451] := 16#D1E7;
   // UNICODE_TO_GBK[8452] := 16#5BB5;
   // UNICODE_TO_GBK[8453] := 16#CFFC;
   // UNICODE_TO_GBK[8454] := 16#5BB6;
   // UNICODE_TO_GBK[8455] := 16#BCD2;
   // UNICODE_TO_GBK[8456] := 16#5BB7;
   // UNICODE_TO_GBK[8457] := 16#8C71;
   // UNICODE_TO_GBK[8458] := 16#5BB8;
   // UNICODE_TO_GBK[8459] := 16#E5B7;
   // UNICODE_TO_GBK[8460] := 16#5BB9;
   // UNICODE_TO_GBK[8461] := 16#C8DD;
   // UNICODE_TO_GBK[8462] := 16#5BBA;
   // UNICODE_TO_GBK[8463] := 16#8C72;
   // UNICODE_TO_GBK[8464] := 16#5BBB;
   // UNICODE_TO_GBK[8465] := 16#8C73;
   // UNICODE_TO_GBK[8466] := 16#5BBC;
   // UNICODE_TO_GBK[8467] := 16#8C74;
   // UNICODE_TO_GBK[8468] := 16#5BBD;
   // UNICODE_TO_GBK[8469] := 16#BFED;
   // UNICODE_TO_GBK[8470] := 16#5BBE;
   // UNICODE_TO_GBK[8471] := 16#B1F6;
   // UNICODE_TO_GBK[8472] := 16#5BBF;
   // UNICODE_TO_GBK[8473] := 16#CBDE;
   // UNICODE_TO_GBK[8474] := 16#5BC0;
   // UNICODE_TO_GBK[8475] := 16#8C75;
   // UNICODE_TO_GBK[8476] := 16#5BC1;
   // UNICODE_TO_GBK[8477] := 16#8C76;
   // UNICODE_TO_GBK[8478] := 16#5BC2;
   // UNICODE_TO_GBK[8479] := 16#BCC5;
   // UNICODE_TO_GBK[8480] := 16#5BC3;
   // UNICODE_TO_GBK[8481] := 16#8C77;
   // UNICODE_TO_GBK[8482] := 16#5BC4;
   // UNICODE_TO_GBK[8483] := 16#BCC4;
   // UNICODE_TO_GBK[8484] := 16#5BC5;
   // UNICODE_TO_GBK[8485] := 16#D2FA;
   // UNICODE_TO_GBK[8486] := 16#5BC6;
   // UNICODE_TO_GBK[8487] := 16#C3DC;
   // UNICODE_TO_GBK[8488] := 16#5BC7;
   // UNICODE_TO_GBK[8489] := 16#BFDC;
   // UNICODE_TO_GBK[8490] := 16#5BC8;
   // UNICODE_TO_GBK[8491] := 16#8C78;
   // UNICODE_TO_GBK[8492] := 16#5BC9;
   // UNICODE_TO_GBK[8493] := 16#8C79;
   // UNICODE_TO_GBK[8494] := 16#5BCA;
   // UNICODE_TO_GBK[8495] := 16#8C7A;
   // UNICODE_TO_GBK[8496] := 16#5BCB;
   // UNICODE_TO_GBK[8497] := 16#8C7B;
   // UNICODE_TO_GBK[8498] := 16#5BCC;
   // UNICODE_TO_GBK[8499] := 16#B8BB;
   // UNICODE_TO_GBK[8500] := 16#5BCD;
   // UNICODE_TO_GBK[8501] := 16#8C7C;
   // UNICODE_TO_GBK[8502] := 16#5BCE;
   // UNICODE_TO_GBK[8503] := 16#8C7D;
   // UNICODE_TO_GBK[8504] := 16#5BCF;
   // UNICODE_TO_GBK[8505] := 16#8C7E;
   // UNICODE_TO_GBK[8506] := 16#5BD0;
   // UNICODE_TO_GBK[8507] := 16#C3C2;
   // UNICODE_TO_GBK[8508] := 16#5BD1;
   // UNICODE_TO_GBK[8509] := 16#8C80;
   // UNICODE_TO_GBK[8510] := 16#5BD2;
   // UNICODE_TO_GBK[8511] := 16#BAAE;
   // UNICODE_TO_GBK[8512] := 16#5BD3;
   // UNICODE_TO_GBK[8513] := 16#D4A2;
   // UNICODE_TO_GBK[8514] := 16#5BD4;
   // UNICODE_TO_GBK[8515] := 16#8C81;
   // UNICODE_TO_GBK[8516] := 16#5BD5;
   // UNICODE_TO_GBK[8517] := 16#8C82;
   // UNICODE_TO_GBK[8518] := 16#5BD6;
   // UNICODE_TO_GBK[8519] := 16#8C83;
   // UNICODE_TO_GBK[8520] := 16#5BD7;
   // UNICODE_TO_GBK[8521] := 16#8C84;
   // UNICODE_TO_GBK[8522] := 16#5BD8;
   // UNICODE_TO_GBK[8523] := 16#8C85;
   // UNICODE_TO_GBK[8524] := 16#5BD9;
   // UNICODE_TO_GBK[8525] := 16#8C86;
   // UNICODE_TO_GBK[8526] := 16#5BDA;
   // UNICODE_TO_GBK[8527] := 16#8C87;
   // UNICODE_TO_GBK[8528] := 16#5BDB;
   // UNICODE_TO_GBK[8529] := 16#8C88;
   // UNICODE_TO_GBK[8530] := 16#5BDC;
   // UNICODE_TO_GBK[8531] := 16#8C89;
   // UNICODE_TO_GBK[8532] := 16#5BDD;
   // UNICODE_TO_GBK[8533] := 16#C7DE;
   // UNICODE_TO_GBK[8534] := 16#5BDE;
   // UNICODE_TO_GBK[8535] := 16#C4AF;
   // UNICODE_TO_GBK[8536] := 16#5BDF;
   // UNICODE_TO_GBK[8537] := 16#B2EC;
   // UNICODE_TO_GBK[8538] := 16#5BE0;
   // UNICODE_TO_GBK[8539] := 16#8C8A;
   // UNICODE_TO_GBK[8540] := 16#5BE1;
   // UNICODE_TO_GBK[8541] := 16#B9D1;
   // UNICODE_TO_GBK[8542] := 16#5BE2;
   // UNICODE_TO_GBK[8543] := 16#8C8B;
   // UNICODE_TO_GBK[8544] := 16#5BE3;
   // UNICODE_TO_GBK[8545] := 16#8C8C;
   // UNICODE_TO_GBK[8546] := 16#5BE4;
   // UNICODE_TO_GBK[8547] := 16#E5BB;
   // UNICODE_TO_GBK[8548] := 16#5BE5;
   // UNICODE_TO_GBK[8549] := 16#C1C8;
   // UNICODE_TO_GBK[8550] := 16#5BE6;
   // UNICODE_TO_GBK[8551] := 16#8C8D;
   // UNICODE_TO_GBK[8552] := 16#5BE7;
   // UNICODE_TO_GBK[8553] := 16#8C8E;
   // UNICODE_TO_GBK[8554] := 16#5BE8;
   // UNICODE_TO_GBK[8555] := 16#D5AF;
   // UNICODE_TO_GBK[8556] := 16#5BE9;
   // UNICODE_TO_GBK[8557] := 16#8C8F;
   // UNICODE_TO_GBK[8558] := 16#5BEA;
   // UNICODE_TO_GBK[8559] := 16#8C90;
   // UNICODE_TO_GBK[8560] := 16#5BEB;
   // UNICODE_TO_GBK[8561] := 16#8C91;
   // UNICODE_TO_GBK[8562] := 16#5BEC;
   // UNICODE_TO_GBK[8563] := 16#8C92;
   // UNICODE_TO_GBK[8564] := 16#5BED;
   // UNICODE_TO_GBK[8565] := 16#8C93;
   // UNICODE_TO_GBK[8566] := 16#5BEE;
   // UNICODE_TO_GBK[8567] := 16#E5BC;
   // UNICODE_TO_GBK[8568] := 16#5BEF;
   // UNICODE_TO_GBK[8569] := 16#8C94;
   // UNICODE_TO_GBK[8570] := 16#5BF0;
   // UNICODE_TO_GBK[8571] := 16#E5BE;
   // UNICODE_TO_GBK[8572] := 16#5BF1;
   // UNICODE_TO_GBK[8573] := 16#8C95;
   // UNICODE_TO_GBK[8574] := 16#5BF2;
   // UNICODE_TO_GBK[8575] := 16#8C96;
   // UNICODE_TO_GBK[8576] := 16#5BF3;
   // UNICODE_TO_GBK[8577] := 16#8C97;
   // UNICODE_TO_GBK[8578] := 16#5BF4;
   // UNICODE_TO_GBK[8579] := 16#8C98;
   // UNICODE_TO_GBK[8580] := 16#5BF5;
   // UNICODE_TO_GBK[8581] := 16#8C99;
   // UNICODE_TO_GBK[8582] := 16#5BF6;
   // UNICODE_TO_GBK[8583] := 16#8C9A;
   // UNICODE_TO_GBK[8584] := 16#5BF7;
   // UNICODE_TO_GBK[8585] := 16#8C9B;
   // UNICODE_TO_GBK[8586] := 16#5BF8;
   // UNICODE_TO_GBK[8587] := 16#B4E7;
   // UNICODE_TO_GBK[8588] := 16#5BF9;
   // UNICODE_TO_GBK[8589] := 16#B6D4;
   // UNICODE_TO_GBK[8590] := 16#5BFA;
   // UNICODE_TO_GBK[8591] := 16#CBC2;
   // UNICODE_TO_GBK[8592] := 16#5BFB;
   // UNICODE_TO_GBK[8593] := 16#D1B0;
   // UNICODE_TO_GBK[8594] := 16#5BFC;
   // UNICODE_TO_GBK[8595] := 16#B5BC;
   // UNICODE_TO_GBK[8596] := 16#5BFD;
   // UNICODE_TO_GBK[8597] := 16#8C9C;
   // UNICODE_TO_GBK[8598] := 16#5BFE;
   // UNICODE_TO_GBK[8599] := 16#8C9D;
   // UNICODE_TO_GBK[8600] := 16#5BFF;
   // UNICODE_TO_GBK[8601] := 16#CAD9;
   // UNICODE_TO_GBK[8602] := 16#5C00;
   // UNICODE_TO_GBK[8603] := 16#8C9E;
   // UNICODE_TO_GBK[8604] := 16#5C01;
   // UNICODE_TO_GBK[8605] := 16#B7E2;
   // UNICODE_TO_GBK[8606] := 16#5C02;
   // UNICODE_TO_GBK[8607] := 16#8C9F;
   // UNICODE_TO_GBK[8608] := 16#5C03;
   // UNICODE_TO_GBK[8609] := 16#8CA0;
   // UNICODE_TO_GBK[8610] := 16#5C04;
   // UNICODE_TO_GBK[8611] := 16#C9E4;
   // UNICODE_TO_GBK[8612] := 16#5C05;
   // UNICODE_TO_GBK[8613] := 16#8CA1;
   // UNICODE_TO_GBK[8614] := 16#5C06;
   // UNICODE_TO_GBK[8615] := 16#BDAB;
   // UNICODE_TO_GBK[8616] := 16#5C07;
   // UNICODE_TO_GBK[8617] := 16#8CA2;
   // UNICODE_TO_GBK[8618] := 16#5C08;
   // UNICODE_TO_GBK[8619] := 16#8CA3;
   // UNICODE_TO_GBK[8620] := 16#5C09;
   // UNICODE_TO_GBK[8621] := 16#CEBE;
   // UNICODE_TO_GBK[8622] := 16#5C0A;
   // UNICODE_TO_GBK[8623] := 16#D7F0;
   // UNICODE_TO_GBK[8624] := 16#5C0B;
   // UNICODE_TO_GBK[8625] := 16#8CA4;
   // UNICODE_TO_GBK[8626] := 16#5C0C;
   // UNICODE_TO_GBK[8627] := 16#8CA5;
   // UNICODE_TO_GBK[8628] := 16#5C0D;
   // UNICODE_TO_GBK[8629] := 16#8CA6;
   // UNICODE_TO_GBK[8630] := 16#5C0E;
   // UNICODE_TO_GBK[8631] := 16#8CA7;
   // UNICODE_TO_GBK[8632] := 16#5C0F;
   // UNICODE_TO_GBK[8633] := 16#D0A1;
   // UNICODE_TO_GBK[8634] := 16#5C10;
   // UNICODE_TO_GBK[8635] := 16#8CA8;
   // UNICODE_TO_GBK[8636] := 16#5C11;
   // UNICODE_TO_GBK[8637] := 16#C9D9;
   // UNICODE_TO_GBK[8638] := 16#5C12;
   // UNICODE_TO_GBK[8639] := 16#8CA9;
   // UNICODE_TO_GBK[8640] := 16#5C13;
   // UNICODE_TO_GBK[8641] := 16#8CAA;
   // UNICODE_TO_GBK[8642] := 16#5C14;
   // UNICODE_TO_GBK[8643] := 16#B6FB;
   // UNICODE_TO_GBK[8644] := 16#5C15;
   // UNICODE_TO_GBK[8645] := 16#E6D8;
   // UNICODE_TO_GBK[8646] := 16#5C16;
   // UNICODE_TO_GBK[8647] := 16#BCE2;
   // UNICODE_TO_GBK[8648] := 16#5C17;
   // UNICODE_TO_GBK[8649] := 16#8CAB;
   // UNICODE_TO_GBK[8650] := 16#5C18;
   // UNICODE_TO_GBK[8651] := 16#B3BE;
   // UNICODE_TO_GBK[8652] := 16#5C19;
   // UNICODE_TO_GBK[8653] := 16#8CAC;
   // UNICODE_TO_GBK[8654] := 16#5C1A;
   // UNICODE_TO_GBK[8655] := 16#C9D0;
   // UNICODE_TO_GBK[8656] := 16#5C1B;
   // UNICODE_TO_GBK[8657] := 16#8CAD;
   // UNICODE_TO_GBK[8658] := 16#5C1C;
   // UNICODE_TO_GBK[8659] := 16#E6D9;
   // UNICODE_TO_GBK[8660] := 16#5C1D;
   // UNICODE_TO_GBK[8661] := 16#B3A2;
   // UNICODE_TO_GBK[8662] := 16#5C1E;
   // UNICODE_TO_GBK[8663] := 16#8CAE;
   // UNICODE_TO_GBK[8664] := 16#5C1F;
   // UNICODE_TO_GBK[8665] := 16#8CAF;
   // UNICODE_TO_GBK[8666] := 16#5C20;
   // UNICODE_TO_GBK[8667] := 16#8CB0;
   // UNICODE_TO_GBK[8668] := 16#5C21;
   // UNICODE_TO_GBK[8669] := 16#8CB1;
   // UNICODE_TO_GBK[8670] := 16#5C22;
   // UNICODE_TO_GBK[8671] := 16#DECC;
   // UNICODE_TO_GBK[8672] := 16#5C23;
   // UNICODE_TO_GBK[8673] := 16#8CB2;
   // UNICODE_TO_GBK[8674] := 16#5C24;
   // UNICODE_TO_GBK[8675] := 16#D3C8;
   // UNICODE_TO_GBK[8676] := 16#5C25;
   // UNICODE_TO_GBK[8677] := 16#DECD;
   // UNICODE_TO_GBK[8678] := 16#5C26;
   // UNICODE_TO_GBK[8679] := 16#8CB3;
   // UNICODE_TO_GBK[8680] := 16#5C27;
   // UNICODE_TO_GBK[8681] := 16#D2A2;
   // UNICODE_TO_GBK[8682] := 16#5C28;
   // UNICODE_TO_GBK[8683] := 16#8CB4;
   // UNICODE_TO_GBK[8684] := 16#5C29;
   // UNICODE_TO_GBK[8685] := 16#8CB5;
   // UNICODE_TO_GBK[8686] := 16#5C2A;
   // UNICODE_TO_GBK[8687] := 16#8CB6;
   // UNICODE_TO_GBK[8688] := 16#5C2B;
   // UNICODE_TO_GBK[8689] := 16#8CB7;
   // UNICODE_TO_GBK[8690] := 16#5C2C;
   // UNICODE_TO_GBK[8691] := 16#DECE;
   // UNICODE_TO_GBK[8692] := 16#5C2D;
   // UNICODE_TO_GBK[8693] := 16#8CB8;
   // UNICODE_TO_GBK[8694] := 16#5C2E;
   // UNICODE_TO_GBK[8695] := 16#8CB9;
   // UNICODE_TO_GBK[8696] := 16#5C2F;
   // UNICODE_TO_GBK[8697] := 16#8CBA;
   // UNICODE_TO_GBK[8698] := 16#5C30;
   // UNICODE_TO_GBK[8699] := 16#8CBB;
   // UNICODE_TO_GBK[8700] := 16#5C31;
   // UNICODE_TO_GBK[8701] := 16#BECD;
   // UNICODE_TO_GBK[8702] := 16#5C32;
   // UNICODE_TO_GBK[8703] := 16#8CBC;
   // UNICODE_TO_GBK[8704] := 16#5C33;
   // UNICODE_TO_GBK[8705] := 16#8CBD;
   // UNICODE_TO_GBK[8706] := 16#5C34;
   // UNICODE_TO_GBK[8707] := 16#DECF;
   // UNICODE_TO_GBK[8708] := 16#5C35;
   // UNICODE_TO_GBK[8709] := 16#8CBE;
   // UNICODE_TO_GBK[8710] := 16#5C36;
   // UNICODE_TO_GBK[8711] := 16#8CBF;
   // UNICODE_TO_GBK[8712] := 16#5C37;
   // UNICODE_TO_GBK[8713] := 16#8CC0;
   // UNICODE_TO_GBK[8714] := 16#5C38;
   // UNICODE_TO_GBK[8715] := 16#CAAC;
   // UNICODE_TO_GBK[8716] := 16#5C39;
   // UNICODE_TO_GBK[8717] := 16#D2FC;
   // UNICODE_TO_GBK[8718] := 16#5C3A;
   // UNICODE_TO_GBK[8719] := 16#B3DF;
   // UNICODE_TO_GBK[8720] := 16#5C3B;
   // UNICODE_TO_GBK[8721] := 16#E5EA;
   // UNICODE_TO_GBK[8722] := 16#5C3C;
   // UNICODE_TO_GBK[8723] := 16#C4E1;
   // UNICODE_TO_GBK[8724] := 16#5C3D;
   // UNICODE_TO_GBK[8725] := 16#BEA1;
   // UNICODE_TO_GBK[8726] := 16#5C3E;
   // UNICODE_TO_GBK[8727] := 16#CEB2;
   // UNICODE_TO_GBK[8728] := 16#5C3F;
   // UNICODE_TO_GBK[8729] := 16#C4F2;
   // UNICODE_TO_GBK[8730] := 16#5C40;
   // UNICODE_TO_GBK[8731] := 16#BED6;
   // UNICODE_TO_GBK[8732] := 16#5C41;
   // UNICODE_TO_GBK[8733] := 16#C6A8;
   // UNICODE_TO_GBK[8734] := 16#5C42;
   // UNICODE_TO_GBK[8735] := 16#B2E3;
   // UNICODE_TO_GBK[8736] := 16#5C43;
   // UNICODE_TO_GBK[8737] := 16#8CC1;
   // UNICODE_TO_GBK[8738] := 16#5C44;
   // UNICODE_TO_GBK[8739] := 16#8CC2;
   // UNICODE_TO_GBK[8740] := 16#5C45;
   // UNICODE_TO_GBK[8741] := 16#BED3;
   // UNICODE_TO_GBK[8742] := 16#5C46;
   // UNICODE_TO_GBK[8743] := 16#8CC3;
   // UNICODE_TO_GBK[8744] := 16#5C47;
   // UNICODE_TO_GBK[8745] := 16#8CC4;
   // UNICODE_TO_GBK[8746] := 16#5C48;
   // UNICODE_TO_GBK[8747] := 16#C7FC;
   // UNICODE_TO_GBK[8748] := 16#5C49;
   // UNICODE_TO_GBK[8749] := 16#CCEB;
   // UNICODE_TO_GBK[8750] := 16#5C4A;
   // UNICODE_TO_GBK[8751] := 16#BDEC;
   // UNICODE_TO_GBK[8752] := 16#5C4B;
   // UNICODE_TO_GBK[8753] := 16#CEDD;
   // UNICODE_TO_GBK[8754] := 16#5C4C;
   // UNICODE_TO_GBK[8755] := 16#8CC5;
   // UNICODE_TO_GBK[8756] := 16#5C4D;
   // UNICODE_TO_GBK[8757] := 16#8CC6;
   // UNICODE_TO_GBK[8758] := 16#5C4E;
   // UNICODE_TO_GBK[8759] := 16#CABA;
   // UNICODE_TO_GBK[8760] := 16#5C4F;
   // UNICODE_TO_GBK[8761] := 16#C6C1;
   // UNICODE_TO_GBK[8762] := 16#5C50;
   // UNICODE_TO_GBK[8763] := 16#E5EC;
   // UNICODE_TO_GBK[8764] := 16#5C51;
   // UNICODE_TO_GBK[8765] := 16#D0BC;
   // UNICODE_TO_GBK[8766] := 16#5C52;
   // UNICODE_TO_GBK[8767] := 16#8CC7;
   // UNICODE_TO_GBK[8768] := 16#5C53;
   // UNICODE_TO_GBK[8769] := 16#8CC8;
   // UNICODE_TO_GBK[8770] := 16#5C54;
   // UNICODE_TO_GBK[8771] := 16#8CC9;
   // UNICODE_TO_GBK[8772] := 16#5C55;
   // UNICODE_TO_GBK[8773] := 16#D5B9;
   // UNICODE_TO_GBK[8774] := 16#5C56;
   // UNICODE_TO_GBK[8775] := 16#8CCA;
   // UNICODE_TO_GBK[8776] := 16#5C57;
   // UNICODE_TO_GBK[8777] := 16#8CCB;
   // UNICODE_TO_GBK[8778] := 16#5C58;
   // UNICODE_TO_GBK[8779] := 16#8CCC;
   // UNICODE_TO_GBK[8780] := 16#5C59;
   // UNICODE_TO_GBK[8781] := 16#E5ED;
   // UNICODE_TO_GBK[8782] := 16#5C5A;
   // UNICODE_TO_GBK[8783] := 16#8CCD;
   // UNICODE_TO_GBK[8784] := 16#5C5B;
   // UNICODE_TO_GBK[8785] := 16#8CCE;
   // UNICODE_TO_GBK[8786] := 16#5C5C;
   // UNICODE_TO_GBK[8787] := 16#8CCF;
   // UNICODE_TO_GBK[8788] := 16#5C5D;
   // UNICODE_TO_GBK[8789] := 16#8CD0;
   // UNICODE_TO_GBK[8790] := 16#5C5E;
   // UNICODE_TO_GBK[8791] := 16#CAF4;
   // UNICODE_TO_GBK[8792] := 16#5C5F;
   // UNICODE_TO_GBK[8793] := 16#8CD1;
   // UNICODE_TO_GBK[8794] := 16#5C60;
   // UNICODE_TO_GBK[8795] := 16#CDC0;
   // UNICODE_TO_GBK[8796] := 16#5C61;
   // UNICODE_TO_GBK[8797] := 16#C2C5;
   // UNICODE_TO_GBK[8798] := 16#5C62;
   // UNICODE_TO_GBK[8799] := 16#8CD2;
   // UNICODE_TO_GBK[8800] := 16#5C63;
   // UNICODE_TO_GBK[8801] := 16#E5EF;
   // UNICODE_TO_GBK[8802] := 16#5C64;
   // UNICODE_TO_GBK[8803] := 16#8CD3;
   // UNICODE_TO_GBK[8804] := 16#5C65;
   // UNICODE_TO_GBK[8805] := 16#C2C4;
   // UNICODE_TO_GBK[8806] := 16#5C66;
   // UNICODE_TO_GBK[8807] := 16#E5F0;
   // UNICODE_TO_GBK[8808] := 16#5C67;
   // UNICODE_TO_GBK[8809] := 16#8CD4;
   // UNICODE_TO_GBK[8810] := 16#5C68;
   // UNICODE_TO_GBK[8811] := 16#8CD5;
   // UNICODE_TO_GBK[8812] := 16#5C69;
   // UNICODE_TO_GBK[8813] := 16#8CD6;
   // UNICODE_TO_GBK[8814] := 16#5C6A;
   // UNICODE_TO_GBK[8815] := 16#8CD7;
   // UNICODE_TO_GBK[8816] := 16#5C6B;
   // UNICODE_TO_GBK[8817] := 16#8CD8;
   // UNICODE_TO_GBK[8818] := 16#5C6C;
   // UNICODE_TO_GBK[8819] := 16#8CD9;
   // UNICODE_TO_GBK[8820] := 16#5C6D;
   // UNICODE_TO_GBK[8821] := 16#8CDA;
   // UNICODE_TO_GBK[8822] := 16#5C6E;
   // UNICODE_TO_GBK[8823] := 16#E5F8;
   // UNICODE_TO_GBK[8824] := 16#5C6F;
   // UNICODE_TO_GBK[8825] := 16#CDCD;
   // UNICODE_TO_GBK[8826] := 16#5C70;
   // UNICODE_TO_GBK[8827] := 16#8CDB;
   // UNICODE_TO_GBK[8828] := 16#5C71;
   // UNICODE_TO_GBK[8829] := 16#C9BD;
   // UNICODE_TO_GBK[8830] := 16#5C72;
   // UNICODE_TO_GBK[8831] := 16#8CDC;
   // UNICODE_TO_GBK[8832] := 16#5C73;
   // UNICODE_TO_GBK[8833] := 16#8CDD;
   // UNICODE_TO_GBK[8834] := 16#5C74;
   // UNICODE_TO_GBK[8835] := 16#8CDE;
   // UNICODE_TO_GBK[8836] := 16#5C75;
   // UNICODE_TO_GBK[8837] := 16#8CDF;
   // UNICODE_TO_GBK[8838] := 16#5C76;
   // UNICODE_TO_GBK[8839] := 16#8CE0;
   // UNICODE_TO_GBK[8840] := 16#5C77;
   // UNICODE_TO_GBK[8841] := 16#8CE1;
   // UNICODE_TO_GBK[8842] := 16#5C78;
   // UNICODE_TO_GBK[8843] := 16#8CE2;
   // UNICODE_TO_GBK[8844] := 16#5C79;
   // UNICODE_TO_GBK[8845] := 16#D2D9;
   // UNICODE_TO_GBK[8846] := 16#5C7A;
   // UNICODE_TO_GBK[8847] := 16#E1A8;
   // UNICODE_TO_GBK[8848] := 16#5C7B;
   // UNICODE_TO_GBK[8849] := 16#8CE3;
   // UNICODE_TO_GBK[8850] := 16#5C7C;
   // UNICODE_TO_GBK[8851] := 16#8CE4;
   // UNICODE_TO_GBK[8852] := 16#5C7D;
   // UNICODE_TO_GBK[8853] := 16#8CE5;
   // UNICODE_TO_GBK[8854] := 16#5C7E;
   // UNICODE_TO_GBK[8855] := 16#8CE6;
   // UNICODE_TO_GBK[8856] := 16#5C7F;
   // UNICODE_TO_GBK[8857] := 16#D3EC;
   // UNICODE_TO_GBK[8858] := 16#5C80;
   // UNICODE_TO_GBK[8859] := 16#8CE7;
   // UNICODE_TO_GBK[8860] := 16#5C81;
   // UNICODE_TO_GBK[8861] := 16#CBEA;
   // UNICODE_TO_GBK[8862] := 16#5C82;
   // UNICODE_TO_GBK[8863] := 16#C6F1;
   // UNICODE_TO_GBK[8864] := 16#5C83;
   // UNICODE_TO_GBK[8865] := 16#8CE8;
   // UNICODE_TO_GBK[8866] := 16#5C84;
   // UNICODE_TO_GBK[8867] := 16#8CE9;
   // UNICODE_TO_GBK[8868] := 16#5C85;
   // UNICODE_TO_GBK[8869] := 16#8CEA;
   // UNICODE_TO_GBK[8870] := 16#5C86;
   // UNICODE_TO_GBK[8871] := 16#8CEB;
   // UNICODE_TO_GBK[8872] := 16#5C87;
   // UNICODE_TO_GBK[8873] := 16#8CEC;
   // UNICODE_TO_GBK[8874] := 16#5C88;
   // UNICODE_TO_GBK[8875] := 16#E1AC;
   // UNICODE_TO_GBK[8876] := 16#5C89;
   // UNICODE_TO_GBK[8877] := 16#8CED;
   // UNICODE_TO_GBK[8878] := 16#5C8A;
   // UNICODE_TO_GBK[8879] := 16#8CEE;
   // UNICODE_TO_GBK[8880] := 16#5C8B;
   // UNICODE_TO_GBK[8881] := 16#8CEF;
   // UNICODE_TO_GBK[8882] := 16#5C8C;
   // UNICODE_TO_GBK[8883] := 16#E1A7;
   // UNICODE_TO_GBK[8884] := 16#5C8D;
   // UNICODE_TO_GBK[8885] := 16#E1A9;
   // UNICODE_TO_GBK[8886] := 16#5C8E;
   // UNICODE_TO_GBK[8887] := 16#8CF0;
   // UNICODE_TO_GBK[8888] := 16#5C8F;
   // UNICODE_TO_GBK[8889] := 16#8CF1;
   // UNICODE_TO_GBK[8890] := 16#5C90;
   // UNICODE_TO_GBK[8891] := 16#E1AA;
   // UNICODE_TO_GBK[8892] := 16#5C91;
   // UNICODE_TO_GBK[8893] := 16#E1AF;
   // UNICODE_TO_GBK[8894] := 16#5C92;
   // UNICODE_TO_GBK[8895] := 16#8CF2;
   // UNICODE_TO_GBK[8896] := 16#5C93;
   // UNICODE_TO_GBK[8897] := 16#8CF3;
   // UNICODE_TO_GBK[8898] := 16#5C94;
   // UNICODE_TO_GBK[8899] := 16#B2ED;
   // UNICODE_TO_GBK[8900] := 16#5C95;
   // UNICODE_TO_GBK[8901] := 16#8CF4;
   // UNICODE_TO_GBK[8902] := 16#5C96;
   // UNICODE_TO_GBK[8903] := 16#E1AB;
   // UNICODE_TO_GBK[8904] := 16#5C97;
   // UNICODE_TO_GBK[8905] := 16#B8DA;
   // UNICODE_TO_GBK[8906] := 16#5C98;
   // UNICODE_TO_GBK[8907] := 16#E1AD;
   // UNICODE_TO_GBK[8908] := 16#5C99;
   // UNICODE_TO_GBK[8909] := 16#E1AE;
   // UNICODE_TO_GBK[8910] := 16#5C9A;
   // UNICODE_TO_GBK[8911] := 16#E1B0;
   // UNICODE_TO_GBK[8912] := 16#5C9B;
   // UNICODE_TO_GBK[8913] := 16#B5BA;
   // UNICODE_TO_GBK[8914] := 16#5C9C;
   // UNICODE_TO_GBK[8915] := 16#E1B1;
   // UNICODE_TO_GBK[8916] := 16#5C9D;
   // UNICODE_TO_GBK[8917] := 16#8CF5;
   // UNICODE_TO_GBK[8918] := 16#5C9E;
   // UNICODE_TO_GBK[8919] := 16#8CF6;
   // UNICODE_TO_GBK[8920] := 16#5C9F;
   // UNICODE_TO_GBK[8921] := 16#8CF7;
   // UNICODE_TO_GBK[8922] := 16#5CA0;
   // UNICODE_TO_GBK[8923] := 16#8CF8;
   // UNICODE_TO_GBK[8924] := 16#5CA1;
   // UNICODE_TO_GBK[8925] := 16#8CF9;
   // UNICODE_TO_GBK[8926] := 16#5CA2;
   // UNICODE_TO_GBK[8927] := 16#E1B3;
   // UNICODE_TO_GBK[8928] := 16#5CA3;
   // UNICODE_TO_GBK[8929] := 16#E1B8;
   // UNICODE_TO_GBK[8930] := 16#5CA4;
   // UNICODE_TO_GBK[8931] := 16#8CFA;
   // UNICODE_TO_GBK[8932] := 16#5CA5;
   // UNICODE_TO_GBK[8933] := 16#8CFB;
   // UNICODE_TO_GBK[8934] := 16#5CA6;
   // UNICODE_TO_GBK[8935] := 16#8CFC;
   // UNICODE_TO_GBK[8936] := 16#5CA7;
   // UNICODE_TO_GBK[8937] := 16#8CFD;
   // UNICODE_TO_GBK[8938] := 16#5CA8;
   // UNICODE_TO_GBK[8939] := 16#8CFE;
   // UNICODE_TO_GBK[8940] := 16#5CA9;
   // UNICODE_TO_GBK[8941] := 16#D1D2;
   // UNICODE_TO_GBK[8942] := 16#5CAA;
   // UNICODE_TO_GBK[8943] := 16#8D40;
   // UNICODE_TO_GBK[8944] := 16#5CAB;
   // UNICODE_TO_GBK[8945] := 16#E1B6;
   // UNICODE_TO_GBK[8946] := 16#5CAC;
   // UNICODE_TO_GBK[8947] := 16#E1B5;
   // UNICODE_TO_GBK[8948] := 16#5CAD;
   // UNICODE_TO_GBK[8949] := 16#C1EB;
   // UNICODE_TO_GBK[8950] := 16#5CAE;
   // UNICODE_TO_GBK[8951] := 16#8D41;
   // UNICODE_TO_GBK[8952] := 16#5CAF;
   // UNICODE_TO_GBK[8953] := 16#8D42;
   // UNICODE_TO_GBK[8954] := 16#5CB0;
   // UNICODE_TO_GBK[8955] := 16#8D43;
   // UNICODE_TO_GBK[8956] := 16#5CB1;
   // UNICODE_TO_GBK[8957] := 16#E1B7;
   // UNICODE_TO_GBK[8958] := 16#5CB2;
   // UNICODE_TO_GBK[8959] := 16#8D44;
   // UNICODE_TO_GBK[8960] := 16#5CB3;
   // UNICODE_TO_GBK[8961] := 16#D4C0;
   // UNICODE_TO_GBK[8962] := 16#5CB4;
   // UNICODE_TO_GBK[8963] := 16#8D45;
   // UNICODE_TO_GBK[8964] := 16#5CB5;
   // UNICODE_TO_GBK[8965] := 16#E1B2;
   // UNICODE_TO_GBK[8966] := 16#5CB6;
   // UNICODE_TO_GBK[8967] := 16#8D46;
   // UNICODE_TO_GBK[8968] := 16#5CB7;
   // UNICODE_TO_GBK[8969] := 16#E1BA;
   // UNICODE_TO_GBK[8970] := 16#5CB8;
   // UNICODE_TO_GBK[8971] := 16#B0B6;
   // UNICODE_TO_GBK[8972] := 16#5CB9;
   // UNICODE_TO_GBK[8973] := 16#8D47;
   // UNICODE_TO_GBK[8974] := 16#5CBA;
   // UNICODE_TO_GBK[8975] := 16#8D48;
   // UNICODE_TO_GBK[8976] := 16#5CBB;
   // UNICODE_TO_GBK[8977] := 16#8D49;
   // UNICODE_TO_GBK[8978] := 16#5CBC;
   // UNICODE_TO_GBK[8979] := 16#8D4A;
   // UNICODE_TO_GBK[8980] := 16#5CBD;
   // UNICODE_TO_GBK[8981] := 16#E1B4;
   // UNICODE_TO_GBK[8982] := 16#5CBE;
   // UNICODE_TO_GBK[8983] := 16#8D4B;
   // UNICODE_TO_GBK[8984] := 16#5CBF;
   // UNICODE_TO_GBK[8985] := 16#BFF9;
   // UNICODE_TO_GBK[8986] := 16#5CC0;
   // UNICODE_TO_GBK[8987] := 16#8D4C;
   // UNICODE_TO_GBK[8988] := 16#5CC1;
   // UNICODE_TO_GBK[8989] := 16#E1B9;
   // UNICODE_TO_GBK[8990] := 16#5CC2;
   // UNICODE_TO_GBK[8991] := 16#8D4D;
   // UNICODE_TO_GBK[8992] := 16#5CC3;
   // UNICODE_TO_GBK[8993] := 16#8D4E;
   // UNICODE_TO_GBK[8994] := 16#5CC4;
   // UNICODE_TO_GBK[8995] := 16#E1BB;
   // UNICODE_TO_GBK[8996] := 16#5CC5;
   // UNICODE_TO_GBK[8997] := 16#8D4F;
   // UNICODE_TO_GBK[8998] := 16#5CC6;
   // UNICODE_TO_GBK[8999] := 16#8D50;
   // UNICODE_TO_GBK[9000] := 16#5CC7;
   // UNICODE_TO_GBK[9001] := 16#8D51;
   // UNICODE_TO_GBK[9002] := 16#5CC8;
   // UNICODE_TO_GBK[9003] := 16#8D52;
   // UNICODE_TO_GBK[9004] := 16#5CC9;
   // UNICODE_TO_GBK[9005] := 16#8D53;
   // UNICODE_TO_GBK[9006] := 16#5CCA;
   // UNICODE_TO_GBK[9007] := 16#8D54;
   // UNICODE_TO_GBK[9008] := 16#5CCB;
   // UNICODE_TO_GBK[9009] := 16#E1BE;
   // UNICODE_TO_GBK[9010] := 16#5CCC;
   // UNICODE_TO_GBK[9011] := 16#8D55;
   // UNICODE_TO_GBK[9012] := 16#5CCD;
   // UNICODE_TO_GBK[9013] := 16#8D56;
   // UNICODE_TO_GBK[9014] := 16#5CCE;
   // UNICODE_TO_GBK[9015] := 16#8D57;
   // UNICODE_TO_GBK[9016] := 16#5CCF;
   // UNICODE_TO_GBK[9017] := 16#8D58;
   // UNICODE_TO_GBK[9018] := 16#5CD0;
   // UNICODE_TO_GBK[9019] := 16#8D59;
   // UNICODE_TO_GBK[9020] := 16#5CD1;
   // UNICODE_TO_GBK[9021] := 16#8D5A;
   // UNICODE_TO_GBK[9022] := 16#5CD2;
   // UNICODE_TO_GBK[9023] := 16#E1BC;
   // UNICODE_TO_GBK[9024] := 16#5CD3;
   // UNICODE_TO_GBK[9025] := 16#8D5B;
   // UNICODE_TO_GBK[9026] := 16#5CD4;
   // UNICODE_TO_GBK[9027] := 16#8D5C;
   // UNICODE_TO_GBK[9028] := 16#5CD5;
   // UNICODE_TO_GBK[9029] := 16#8D5D;
   // UNICODE_TO_GBK[9030] := 16#5CD6;
   // UNICODE_TO_GBK[9031] := 16#8D5E;
   // UNICODE_TO_GBK[9032] := 16#5CD7;
   // UNICODE_TO_GBK[9033] := 16#8D5F;
   // UNICODE_TO_GBK[9034] := 16#5CD8;
   // UNICODE_TO_GBK[9035] := 16#8D60;
   // UNICODE_TO_GBK[9036] := 16#5CD9;
   // UNICODE_TO_GBK[9037] := 16#D6C5;
   // UNICODE_TO_GBK[9038] := 16#5CDA;
   // UNICODE_TO_GBK[9039] := 16#8D61;
   // UNICODE_TO_GBK[9040] := 16#5CDB;
   // UNICODE_TO_GBK[9041] := 16#8D62;
   // UNICODE_TO_GBK[9042] := 16#5CDC;
   // UNICODE_TO_GBK[9043] := 16#8D63;
   // UNICODE_TO_GBK[9044] := 16#5CDD;
   // UNICODE_TO_GBK[9045] := 16#8D64;
   // UNICODE_TO_GBK[9046] := 16#5CDE;
   // UNICODE_TO_GBK[9047] := 16#8D65;
   // UNICODE_TO_GBK[9048] := 16#5CDF;
   // UNICODE_TO_GBK[9049] := 16#8D66;
   // UNICODE_TO_GBK[9050] := 16#5CE0;
   // UNICODE_TO_GBK[9051] := 16#8D67;
   // UNICODE_TO_GBK[9052] := 16#5CE1;
   // UNICODE_TO_GBK[9053] := 16#CFBF;
   // UNICODE_TO_GBK[9054] := 16#5CE2;
   // UNICODE_TO_GBK[9055] := 16#8D68;
   // UNICODE_TO_GBK[9056] := 16#5CE3;
   // UNICODE_TO_GBK[9057] := 16#8D69;
   // UNICODE_TO_GBK[9058] := 16#5CE4;
   // UNICODE_TO_GBK[9059] := 16#E1BD;
   // UNICODE_TO_GBK[9060] := 16#5CE5;
   // UNICODE_TO_GBK[9061] := 16#E1BF;
   // UNICODE_TO_GBK[9062] := 16#5CE6;
   // UNICODE_TO_GBK[9063] := 16#C2CD;
   // UNICODE_TO_GBK[9064] := 16#5CE7;
   // UNICODE_TO_GBK[9065] := 16#8D6A;
   // UNICODE_TO_GBK[9066] := 16#5CE8;
   // UNICODE_TO_GBK[9067] := 16#B6EB;
   // UNICODE_TO_GBK[9068] := 16#5CE9;
   // UNICODE_TO_GBK[9069] := 16#8D6B;
   // UNICODE_TO_GBK[9070] := 16#5CEA;
   // UNICODE_TO_GBK[9071] := 16#D3F8;
   // UNICODE_TO_GBK[9072] := 16#5CEB;
   // UNICODE_TO_GBK[9073] := 16#8D6C;
   // UNICODE_TO_GBK[9074] := 16#5CEC;
   // UNICODE_TO_GBK[9075] := 16#8D6D;
   // UNICODE_TO_GBK[9076] := 16#5CED;
   // UNICODE_TO_GBK[9077] := 16#C7CD;
   // UNICODE_TO_GBK[9078] := 16#5CEE;
   // UNICODE_TO_GBK[9079] := 16#8D6E;
   // UNICODE_TO_GBK[9080] := 16#5CEF;
   // UNICODE_TO_GBK[9081] := 16#8D6F;
   // UNICODE_TO_GBK[9082] := 16#5CF0;
   // UNICODE_TO_GBK[9083] := 16#B7E5;
   // UNICODE_TO_GBK[9084] := 16#5CF1;
   // UNICODE_TO_GBK[9085] := 16#8D70;
   // UNICODE_TO_GBK[9086] := 16#5CF2;
   // UNICODE_TO_GBK[9087] := 16#8D71;
   // UNICODE_TO_GBK[9088] := 16#5CF3;
   // UNICODE_TO_GBK[9089] := 16#8D72;
   // UNICODE_TO_GBK[9090] := 16#5CF4;
   // UNICODE_TO_GBK[9091] := 16#8D73;
   // UNICODE_TO_GBK[9092] := 16#5CF5;
   // UNICODE_TO_GBK[9093] := 16#8D74;
   // UNICODE_TO_GBK[9094] := 16#5CF6;
   // UNICODE_TO_GBK[9095] := 16#8D75;
   // UNICODE_TO_GBK[9096] := 16#5CF7;
   // UNICODE_TO_GBK[9097] := 16#8D76;
   // UNICODE_TO_GBK[9098] := 16#5CF8;
   // UNICODE_TO_GBK[9099] := 16#8D77;
   // UNICODE_TO_GBK[9100] := 16#5CF9;
   // UNICODE_TO_GBK[9101] := 16#8D78;
   // UNICODE_TO_GBK[9102] := 16#5CFA;
   // UNICODE_TO_GBK[9103] := 16#8D79;
   // UNICODE_TO_GBK[9104] := 16#5CFB;
   // UNICODE_TO_GBK[9105] := 16#BEFE;
   // UNICODE_TO_GBK[9106] := 16#5CFC;
   // UNICODE_TO_GBK[9107] := 16#8D7A;
   // UNICODE_TO_GBK[9108] := 16#5CFD;
   // UNICODE_TO_GBK[9109] := 16#8D7B;
   // UNICODE_TO_GBK[9110] := 16#5CFE;
   // UNICODE_TO_GBK[9111] := 16#8D7C;
   // UNICODE_TO_GBK[9112] := 16#5CFF;
   // UNICODE_TO_GBK[9113] := 16#8D7D;
   // UNICODE_TO_GBK[9114] := 16#5D00;
   // UNICODE_TO_GBK[9115] := 16#8D7E;
   // UNICODE_TO_GBK[9116] := 16#5D01;
   // UNICODE_TO_GBK[9117] := 16#8D80;
   // UNICODE_TO_GBK[9118] := 16#5D02;
   // UNICODE_TO_GBK[9119] := 16#E1C0;
   // UNICODE_TO_GBK[9120] := 16#5D03;
   // UNICODE_TO_GBK[9121] := 16#E1C1;
   // UNICODE_TO_GBK[9122] := 16#5D04;
   // UNICODE_TO_GBK[9123] := 16#8D81;
   // UNICODE_TO_GBK[9124] := 16#5D05;
   // UNICODE_TO_GBK[9125] := 16#8D82;
   // UNICODE_TO_GBK[9126] := 16#5D06;
   // UNICODE_TO_GBK[9127] := 16#E1C7;
   // UNICODE_TO_GBK[9128] := 16#5D07;
   // UNICODE_TO_GBK[9129] := 16#B3E7;
   // UNICODE_TO_GBK[9130] := 16#5D08;
   // UNICODE_TO_GBK[9131] := 16#8D83;
   // UNICODE_TO_GBK[9132] := 16#5D09;
   // UNICODE_TO_GBK[9133] := 16#8D84;
   // UNICODE_TO_GBK[9134] := 16#5D0A;
   // UNICODE_TO_GBK[9135] := 16#8D85;
   // UNICODE_TO_GBK[9136] := 16#5D0B;
   // UNICODE_TO_GBK[9137] := 16#8D86;
   // UNICODE_TO_GBK[9138] := 16#5D0C;
   // UNICODE_TO_GBK[9139] := 16#8D87;
   // UNICODE_TO_GBK[9140] := 16#5D0D;
   // UNICODE_TO_GBK[9141] := 16#8D88;
   // UNICODE_TO_GBK[9142] := 16#5D0E;
   // UNICODE_TO_GBK[9143] := 16#C6E9;
   // UNICODE_TO_GBK[9144] := 16#5D0F;
   // UNICODE_TO_GBK[9145] := 16#8D89;
   // UNICODE_TO_GBK[9146] := 16#5D10;
   // UNICODE_TO_GBK[9147] := 16#8D8A;
   // UNICODE_TO_GBK[9148] := 16#5D11;
   // UNICODE_TO_GBK[9149] := 16#8D8B;
   // UNICODE_TO_GBK[9150] := 16#5D12;
   // UNICODE_TO_GBK[9151] := 16#8D8C;
   // UNICODE_TO_GBK[9152] := 16#5D13;
   // UNICODE_TO_GBK[9153] := 16#8D8D;
   // UNICODE_TO_GBK[9154] := 16#5D14;
   // UNICODE_TO_GBK[9155] := 16#B4DE;
   // UNICODE_TO_GBK[9156] := 16#5D15;
   // UNICODE_TO_GBK[9157] := 16#8D8E;
   // UNICODE_TO_GBK[9158] := 16#5D16;
   // UNICODE_TO_GBK[9159] := 16#D1C2;
   // UNICODE_TO_GBK[9160] := 16#5D17;
   // UNICODE_TO_GBK[9161] := 16#8D8F;
   // UNICODE_TO_GBK[9162] := 16#5D18;
   // UNICODE_TO_GBK[9163] := 16#8D90;
   // UNICODE_TO_GBK[9164] := 16#5D19;
   // UNICODE_TO_GBK[9165] := 16#8D91;
   // UNICODE_TO_GBK[9166] := 16#5D1A;
   // UNICODE_TO_GBK[9167] := 16#8D92;
   // UNICODE_TO_GBK[9168] := 16#5D1B;
   // UNICODE_TO_GBK[9169] := 16#E1C8;
   // UNICODE_TO_GBK[9170] := 16#5D1C;
   // UNICODE_TO_GBK[9171] := 16#8D93;
   // UNICODE_TO_GBK[9172] := 16#5D1D;
   // UNICODE_TO_GBK[9173] := 16#8D94;
   // UNICODE_TO_GBK[9174] := 16#5D1E;
   // UNICODE_TO_GBK[9175] := 16#E1C6;
   // UNICODE_TO_GBK[9176] := 16#5D1F;
   // UNICODE_TO_GBK[9177] := 16#8D95;
   // UNICODE_TO_GBK[9178] := 16#5D20;
   // UNICODE_TO_GBK[9179] := 16#8D96;
   // UNICODE_TO_GBK[9180] := 16#5D21;
   // UNICODE_TO_GBK[9181] := 16#8D97;
   // UNICODE_TO_GBK[9182] := 16#5D22;
   // UNICODE_TO_GBK[9183] := 16#8D98;
   // UNICODE_TO_GBK[9184] := 16#5D23;
   // UNICODE_TO_GBK[9185] := 16#8D99;
   // UNICODE_TO_GBK[9186] := 16#5D24;
   // UNICODE_TO_GBK[9187] := 16#E1C5;
   // UNICODE_TO_GBK[9188] := 16#5D25;
   // UNICODE_TO_GBK[9189] := 16#8D9A;
   // UNICODE_TO_GBK[9190] := 16#5D26;
   // UNICODE_TO_GBK[9191] := 16#E1C3;
   // UNICODE_TO_GBK[9192] := 16#5D27;
   // UNICODE_TO_GBK[9193] := 16#E1C2;
   // UNICODE_TO_GBK[9194] := 16#5D28;
   // UNICODE_TO_GBK[9195] := 16#8D9B;
   // UNICODE_TO_GBK[9196] := 16#5D29;
   // UNICODE_TO_GBK[9197] := 16#B1C0;
   // UNICODE_TO_GBK[9198] := 16#5D2A;
   // UNICODE_TO_GBK[9199] := 16#8D9C;
   // UNICODE_TO_GBK[9200] := 16#5D2B;
   // UNICODE_TO_GBK[9201] := 16#8D9D;
   // UNICODE_TO_GBK[9202] := 16#5D2C;
   // UNICODE_TO_GBK[9203] := 16#8D9E;
   // UNICODE_TO_GBK[9204] := 16#5D2D;
   // UNICODE_TO_GBK[9205] := 16#D5B8;
   // UNICODE_TO_GBK[9206] := 16#5D2E;
   // UNICODE_TO_GBK[9207] := 16#E1C4;
   // UNICODE_TO_GBK[9208] := 16#5D2F;
   // UNICODE_TO_GBK[9209] := 16#8D9F;
   // UNICODE_TO_GBK[9210] := 16#5D30;
   // UNICODE_TO_GBK[9211] := 16#8DA0;
   // UNICODE_TO_GBK[9212] := 16#5D31;
   // UNICODE_TO_GBK[9213] := 16#8DA1;
   // UNICODE_TO_GBK[9214] := 16#5D32;
   // UNICODE_TO_GBK[9215] := 16#8DA2;
   // UNICODE_TO_GBK[9216] := 16#5D33;
   // UNICODE_TO_GBK[9217] := 16#8DA3;
   // UNICODE_TO_GBK[9218] := 16#5D34;
   // UNICODE_TO_GBK[9219] := 16#E1CB;
   // UNICODE_TO_GBK[9220] := 16#5D35;
   // UNICODE_TO_GBK[9221] := 16#8DA4;
   // UNICODE_TO_GBK[9222] := 16#5D36;
   // UNICODE_TO_GBK[9223] := 16#8DA5;
   // UNICODE_TO_GBK[9224] := 16#5D37;
   // UNICODE_TO_GBK[9225] := 16#8DA6;
   // UNICODE_TO_GBK[9226] := 16#5D38;
   // UNICODE_TO_GBK[9227] := 16#8DA7;
   // UNICODE_TO_GBK[9228] := 16#5D39;
   // UNICODE_TO_GBK[9229] := 16#8DA8;
   // UNICODE_TO_GBK[9230] := 16#5D3A;
   // UNICODE_TO_GBK[9231] := 16#8DA9;
   // UNICODE_TO_GBK[9232] := 16#5D3B;
   // UNICODE_TO_GBK[9233] := 16#8DAA;
   // UNICODE_TO_GBK[9234] := 16#5D3C;
   // UNICODE_TO_GBK[9235] := 16#8DAB;
   // UNICODE_TO_GBK[9236] := 16#5D3D;
   // UNICODE_TO_GBK[9237] := 16#E1CC;
   // UNICODE_TO_GBK[9238] := 16#5D3E;
   // UNICODE_TO_GBK[9239] := 16#E1CA;
   // UNICODE_TO_GBK[9240] := 16#5D3F;
   // UNICODE_TO_GBK[9241] := 16#8DAC;
   // UNICODE_TO_GBK[9242] := 16#5D40;
   // UNICODE_TO_GBK[9243] := 16#8DAD;
   // UNICODE_TO_GBK[9244] := 16#5D41;
   // UNICODE_TO_GBK[9245] := 16#8DAE;
   // UNICODE_TO_GBK[9246] := 16#5D42;
   // UNICODE_TO_GBK[9247] := 16#8DAF;
   // UNICODE_TO_GBK[9248] := 16#5D43;
   // UNICODE_TO_GBK[9249] := 16#8DB0;
   // UNICODE_TO_GBK[9250] := 16#5D44;
   // UNICODE_TO_GBK[9251] := 16#8DB1;
   // UNICODE_TO_GBK[9252] := 16#5D45;
   // UNICODE_TO_GBK[9253] := 16#8DB2;
   // UNICODE_TO_GBK[9254] := 16#5D46;
   // UNICODE_TO_GBK[9255] := 16#8DB3;
   // UNICODE_TO_GBK[9256] := 16#5D47;
   // UNICODE_TO_GBK[9257] := 16#EFFA;
   // UNICODE_TO_GBK[9258] := 16#5D48;
   // UNICODE_TO_GBK[9259] := 16#8DB4;
   // UNICODE_TO_GBK[9260] := 16#5D49;
   // UNICODE_TO_GBK[9261] := 16#8DB5;
   // UNICODE_TO_GBK[9262] := 16#5D4A;
   // UNICODE_TO_GBK[9263] := 16#E1D3;
   // UNICODE_TO_GBK[9264] := 16#5D4B;
   // UNICODE_TO_GBK[9265] := 16#E1D2;
   // UNICODE_TO_GBK[9266] := 16#5D4C;
   // UNICODE_TO_GBK[9267] := 16#C7B6;
   // UNICODE_TO_GBK[9268] := 16#5D4D;
   // UNICODE_TO_GBK[9269] := 16#8DB6;
   // UNICODE_TO_GBK[9270] := 16#5D4E;
   // UNICODE_TO_GBK[9271] := 16#8DB7;
   // UNICODE_TO_GBK[9272] := 16#5D4F;
   // UNICODE_TO_GBK[9273] := 16#8DB8;
   // UNICODE_TO_GBK[9274] := 16#5D50;
   // UNICODE_TO_GBK[9275] := 16#8DB9;
   // UNICODE_TO_GBK[9276] := 16#5D51;
   // UNICODE_TO_GBK[9277] := 16#8DBA;
   // UNICODE_TO_GBK[9278] := 16#5D52;
   // UNICODE_TO_GBK[9279] := 16#8DBB;
   // UNICODE_TO_GBK[9280] := 16#5D53;
   // UNICODE_TO_GBK[9281] := 16#8DBC;
   // UNICODE_TO_GBK[9282] := 16#5D54;
   // UNICODE_TO_GBK[9283] := 16#8DBD;
   // UNICODE_TO_GBK[9284] := 16#5D55;
   // UNICODE_TO_GBK[9285] := 16#8DBE;
   // UNICODE_TO_GBK[9286] := 16#5D56;
   // UNICODE_TO_GBK[9287] := 16#8DBF;
   // UNICODE_TO_GBK[9288] := 16#5D57;
   // UNICODE_TO_GBK[9289] := 16#8DC0;
   // UNICODE_TO_GBK[9290] := 16#5D58;
   // UNICODE_TO_GBK[9291] := 16#E1C9;
   // UNICODE_TO_GBK[9292] := 16#5D59;
   // UNICODE_TO_GBK[9293] := 16#8DC1;
   // UNICODE_TO_GBK[9294] := 16#5D5A;
   // UNICODE_TO_GBK[9295] := 16#8DC2;
   // UNICODE_TO_GBK[9296] := 16#5D5B;
   // UNICODE_TO_GBK[9297] := 16#E1CE;
   // UNICODE_TO_GBK[9298] := 16#5D5C;
   // UNICODE_TO_GBK[9299] := 16#8DC3;
   // UNICODE_TO_GBK[9300] := 16#5D5D;
   // UNICODE_TO_GBK[9301] := 16#E1D0;
   // UNICODE_TO_GBK[9302] := 16#5D5E;
   // UNICODE_TO_GBK[9303] := 16#8DC4;
   // UNICODE_TO_GBK[9304] := 16#5D5F;
   // UNICODE_TO_GBK[9305] := 16#8DC5;
   // UNICODE_TO_GBK[9306] := 16#5D60;
   // UNICODE_TO_GBK[9307] := 16#8DC6;
   // UNICODE_TO_GBK[9308] := 16#5D61;
   // UNICODE_TO_GBK[9309] := 16#8DC7;
   // UNICODE_TO_GBK[9310] := 16#5D62;
   // UNICODE_TO_GBK[9311] := 16#8DC8;
   // UNICODE_TO_GBK[9312] := 16#5D63;
   // UNICODE_TO_GBK[9313] := 16#8DC9;
   // UNICODE_TO_GBK[9314] := 16#5D64;
   // UNICODE_TO_GBK[9315] := 16#8DCA;
   // UNICODE_TO_GBK[9316] := 16#5D65;
   // UNICODE_TO_GBK[9317] := 16#8DCB;
   // UNICODE_TO_GBK[9318] := 16#5D66;
   // UNICODE_TO_GBK[9319] := 16#8DCC;
   // UNICODE_TO_GBK[9320] := 16#5D67;
   // UNICODE_TO_GBK[9321] := 16#8DCD;
   // UNICODE_TO_GBK[9322] := 16#5D68;
   // UNICODE_TO_GBK[9323] := 16#8DCE;
   // UNICODE_TO_GBK[9324] := 16#5D69;
   // UNICODE_TO_GBK[9325] := 16#E1D4;
   // UNICODE_TO_GBK[9326] := 16#5D6A;
   // UNICODE_TO_GBK[9327] := 16#8DCF;
   // UNICODE_TO_GBK[9328] := 16#5D6B;
   // UNICODE_TO_GBK[9329] := 16#E1D1;
   // UNICODE_TO_GBK[9330] := 16#5D6C;
   // UNICODE_TO_GBK[9331] := 16#E1CD;
   // UNICODE_TO_GBK[9332] := 16#5D6D;
   // UNICODE_TO_GBK[9333] := 16#8DD0;
   // UNICODE_TO_GBK[9334] := 16#5D6E;
   // UNICODE_TO_GBK[9335] := 16#8DD1;
   // UNICODE_TO_GBK[9336] := 16#5D6F;
   // UNICODE_TO_GBK[9337] := 16#E1CF;
   // UNICODE_TO_GBK[9338] := 16#5D70;
   // UNICODE_TO_GBK[9339] := 16#8DD2;
   // UNICODE_TO_GBK[9340] := 16#5D71;
   // UNICODE_TO_GBK[9341] := 16#8DD3;
   // UNICODE_TO_GBK[9342] := 16#5D72;
   // UNICODE_TO_GBK[9343] := 16#8DD4;
   // UNICODE_TO_GBK[9344] := 16#5D73;
   // UNICODE_TO_GBK[9345] := 16#8DD5;
   // UNICODE_TO_GBK[9346] := 16#5D74;
   // UNICODE_TO_GBK[9347] := 16#E1D5;
   // UNICODE_TO_GBK[9348] := 16#5D75;
   // UNICODE_TO_GBK[9349] := 16#8DD6;
   // UNICODE_TO_GBK[9350] := 16#5D76;
   // UNICODE_TO_GBK[9351] := 16#8DD7;
   // UNICODE_TO_GBK[9352] := 16#5D77;
   // UNICODE_TO_GBK[9353] := 16#8DD8;
   // UNICODE_TO_GBK[9354] := 16#5D78;
   // UNICODE_TO_GBK[9355] := 16#8DD9;
   // UNICODE_TO_GBK[9356] := 16#5D79;
   // UNICODE_TO_GBK[9357] := 16#8DDA;
   // UNICODE_TO_GBK[9358] := 16#5D7A;
   // UNICODE_TO_GBK[9359] := 16#8DDB;
   // UNICODE_TO_GBK[9360] := 16#5D7B;
   // UNICODE_TO_GBK[9361] := 16#8DDC;
   // UNICODE_TO_GBK[9362] := 16#5D7C;
   // UNICODE_TO_GBK[9363] := 16#8DDD;
   // UNICODE_TO_GBK[9364] := 16#5D7D;
   // UNICODE_TO_GBK[9365] := 16#8DDE;
   // UNICODE_TO_GBK[9366] := 16#5D7E;
   // UNICODE_TO_GBK[9367] := 16#8DDF;
   // UNICODE_TO_GBK[9368] := 16#5D7F;
   // UNICODE_TO_GBK[9369] := 16#8DE0;
   // UNICODE_TO_GBK[9370] := 16#5D80;
   // UNICODE_TO_GBK[9371] := 16#8DE1;
   // UNICODE_TO_GBK[9372] := 16#5D81;
   // UNICODE_TO_GBK[9373] := 16#8DE2;
   // UNICODE_TO_GBK[9374] := 16#5D82;
   // UNICODE_TO_GBK[9375] := 16#E1D6;
   // UNICODE_TO_GBK[9376] := 16#5D83;
   // UNICODE_TO_GBK[9377] := 16#8DE3;
   // UNICODE_TO_GBK[9378] := 16#5D84;
   // UNICODE_TO_GBK[9379] := 16#8DE4;
   // UNICODE_TO_GBK[9380] := 16#5D85;
   // UNICODE_TO_GBK[9381] := 16#8DE5;
   // UNICODE_TO_GBK[9382] := 16#5D86;
   // UNICODE_TO_GBK[9383] := 16#8DE6;
   // UNICODE_TO_GBK[9384] := 16#5D87;
   // UNICODE_TO_GBK[9385] := 16#8DE7;
   // UNICODE_TO_GBK[9386] := 16#5D88;
   // UNICODE_TO_GBK[9387] := 16#8DE8;
   // UNICODE_TO_GBK[9388] := 16#5D89;
   // UNICODE_TO_GBK[9389] := 16#8DE9;
   // UNICODE_TO_GBK[9390] := 16#5D8A;
   // UNICODE_TO_GBK[9391] := 16#8DEA;
   // UNICODE_TO_GBK[9392] := 16#5D8B;
   // UNICODE_TO_GBK[9393] := 16#8DEB;
   // UNICODE_TO_GBK[9394] := 16#5D8C;
   // UNICODE_TO_GBK[9395] := 16#8DEC;
   // UNICODE_TO_GBK[9396] := 16#5D8D;
   // UNICODE_TO_GBK[9397] := 16#8DED;
   // UNICODE_TO_GBK[9398] := 16#5D8E;
   // UNICODE_TO_GBK[9399] := 16#8DEE;
   // UNICODE_TO_GBK[9400] := 16#5D8F;
   // UNICODE_TO_GBK[9401] := 16#8DEF;
   // UNICODE_TO_GBK[9402] := 16#5D90;
   // UNICODE_TO_GBK[9403] := 16#8DF0;
   // UNICODE_TO_GBK[9404] := 16#5D91;
   // UNICODE_TO_GBK[9405] := 16#8DF1;
   // UNICODE_TO_GBK[9406] := 16#5D92;
   // UNICODE_TO_GBK[9407] := 16#8DF2;
   // UNICODE_TO_GBK[9408] := 16#5D93;
   // UNICODE_TO_GBK[9409] := 16#8DF3;
   // UNICODE_TO_GBK[9410] := 16#5D94;
   // UNICODE_TO_GBK[9411] := 16#8DF4;
   // UNICODE_TO_GBK[9412] := 16#5D95;
   // UNICODE_TO_GBK[9413] := 16#8DF5;
   // UNICODE_TO_GBK[9414] := 16#5D96;
   // UNICODE_TO_GBK[9415] := 16#8DF6;
   // UNICODE_TO_GBK[9416] := 16#5D97;
   // UNICODE_TO_GBK[9417] := 16#8DF7;
   // UNICODE_TO_GBK[9418] := 16#5D98;
   // UNICODE_TO_GBK[9419] := 16#8DF8;
   // UNICODE_TO_GBK[9420] := 16#5D99;
   // UNICODE_TO_GBK[9421] := 16#E1D7;
   // UNICODE_TO_GBK[9422] := 16#5D9A;
   // UNICODE_TO_GBK[9423] := 16#8DF9;
   // UNICODE_TO_GBK[9424] := 16#5D9B;
   // UNICODE_TO_GBK[9425] := 16#8DFA;
   // UNICODE_TO_GBK[9426] := 16#5D9C;
   // UNICODE_TO_GBK[9427] := 16#8DFB;
   // UNICODE_TO_GBK[9428] := 16#5D9D;
   // UNICODE_TO_GBK[9429] := 16#E1D8;
   // UNICODE_TO_GBK[9430] := 16#5D9E;
   // UNICODE_TO_GBK[9431] := 16#8DFC;
   // UNICODE_TO_GBK[9432] := 16#5D9F;
   // UNICODE_TO_GBK[9433] := 16#8DFD;
   // UNICODE_TO_GBK[9434] := 16#5DA0;
   // UNICODE_TO_GBK[9435] := 16#8DFE;
   // UNICODE_TO_GBK[9436] := 16#5DA1;
   // UNICODE_TO_GBK[9437] := 16#8E40;
   // UNICODE_TO_GBK[9438] := 16#5DA2;
   // UNICODE_TO_GBK[9439] := 16#8E41;
   // UNICODE_TO_GBK[9440] := 16#5DA3;
   // UNICODE_TO_GBK[9441] := 16#8E42;
   // UNICODE_TO_GBK[9442] := 16#5DA4;
   // UNICODE_TO_GBK[9443] := 16#8E43;
   // UNICODE_TO_GBK[9444] := 16#5DA5;
   // UNICODE_TO_GBK[9445] := 16#8E44;
   // UNICODE_TO_GBK[9446] := 16#5DA6;
   // UNICODE_TO_GBK[9447] := 16#8E45;
   // UNICODE_TO_GBK[9448] := 16#5DA7;
   // UNICODE_TO_GBK[9449] := 16#8E46;
   // UNICODE_TO_GBK[9450] := 16#5DA8;
   // UNICODE_TO_GBK[9451] := 16#8E47;
   // UNICODE_TO_GBK[9452] := 16#5DA9;
   // UNICODE_TO_GBK[9453] := 16#8E48;
   // UNICODE_TO_GBK[9454] := 16#5DAA;
   // UNICODE_TO_GBK[9455] := 16#8E49;
   // UNICODE_TO_GBK[9456] := 16#5DAB;
   // UNICODE_TO_GBK[9457] := 16#8E4A;
   // UNICODE_TO_GBK[9458] := 16#5DAC;
   // UNICODE_TO_GBK[9459] := 16#8E4B;
   // UNICODE_TO_GBK[9460] := 16#5DAD;
   // UNICODE_TO_GBK[9461] := 16#8E4C;
   // UNICODE_TO_GBK[9462] := 16#5DAE;
   // UNICODE_TO_GBK[9463] := 16#8E4D;
   // UNICODE_TO_GBK[9464] := 16#5DAF;
   // UNICODE_TO_GBK[9465] := 16#8E4E;
   // UNICODE_TO_GBK[9466] := 16#5DB0;
   // UNICODE_TO_GBK[9467] := 16#8E4F;
   // UNICODE_TO_GBK[9468] := 16#5DB1;
   // UNICODE_TO_GBK[9469] := 16#8E50;
   // UNICODE_TO_GBK[9470] := 16#5DB2;
   // UNICODE_TO_GBK[9471] := 16#8E51;
   // UNICODE_TO_GBK[9472] := 16#5DB3;
   // UNICODE_TO_GBK[9473] := 16#8E52;
   // UNICODE_TO_GBK[9474] := 16#5DB4;
   // UNICODE_TO_GBK[9475] := 16#8E53;
   // UNICODE_TO_GBK[9476] := 16#5DB5;
   // UNICODE_TO_GBK[9477] := 16#8E54;
   // UNICODE_TO_GBK[9478] := 16#5DB6;
   // UNICODE_TO_GBK[9479] := 16#8E55;
   // UNICODE_TO_GBK[9480] := 16#5DB7;
   // UNICODE_TO_GBK[9481] := 16#E1DA;
   // UNICODE_TO_GBK[9482] := 16#5DB8;
   // UNICODE_TO_GBK[9483] := 16#8E56;
   // UNICODE_TO_GBK[9484] := 16#5DB9;
   // UNICODE_TO_GBK[9485] := 16#8E57;
   // UNICODE_TO_GBK[9486] := 16#5DBA;
   // UNICODE_TO_GBK[9487] := 16#8E58;
   // UNICODE_TO_GBK[9488] := 16#5DBB;
   // UNICODE_TO_GBK[9489] := 16#8E59;
   // UNICODE_TO_GBK[9490] := 16#5DBC;
   // UNICODE_TO_GBK[9491] := 16#8E5A;
   // UNICODE_TO_GBK[9492] := 16#5DBD;
   // UNICODE_TO_GBK[9493] := 16#8E5B;
   // UNICODE_TO_GBK[9494] := 16#5DBE;
   // UNICODE_TO_GBK[9495] := 16#8E5C;
   // UNICODE_TO_GBK[9496] := 16#5DBF;
   // UNICODE_TO_GBK[9497] := 16#8E5D;
   // UNICODE_TO_GBK[9498] := 16#5DC0;
   // UNICODE_TO_GBK[9499] := 16#8E5E;
   // UNICODE_TO_GBK[9500] := 16#5DC1;
   // UNICODE_TO_GBK[9501] := 16#8E5F;
   // UNICODE_TO_GBK[9502] := 16#5DC2;
   // UNICODE_TO_GBK[9503] := 16#8E60;
   // UNICODE_TO_GBK[9504] := 16#5DC3;
   // UNICODE_TO_GBK[9505] := 16#8E61;
   // UNICODE_TO_GBK[9506] := 16#5DC4;
   // UNICODE_TO_GBK[9507] := 16#8E62;
   // UNICODE_TO_GBK[9508] := 16#5DC5;
   // UNICODE_TO_GBK[9509] := 16#E1DB;
   // UNICODE_TO_GBK[9510] := 16#5DC6;
   // UNICODE_TO_GBK[9511] := 16#8E63;
   // UNICODE_TO_GBK[9512] := 16#5DC7;
   // UNICODE_TO_GBK[9513] := 16#8E64;
   // UNICODE_TO_GBK[9514] := 16#5DC8;
   // UNICODE_TO_GBK[9515] := 16#8E65;
   // UNICODE_TO_GBK[9516] := 16#5DC9;
   // UNICODE_TO_GBK[9517] := 16#8E66;
   // UNICODE_TO_GBK[9518] := 16#5DCA;
   // UNICODE_TO_GBK[9519] := 16#8E67;
   // UNICODE_TO_GBK[9520] := 16#5DCB;
   // UNICODE_TO_GBK[9521] := 16#8E68;
   // UNICODE_TO_GBK[9522] := 16#5DCC;
   // UNICODE_TO_GBK[9523] := 16#8E69;
   // UNICODE_TO_GBK[9524] := 16#5DCD;
   // UNICODE_TO_GBK[9525] := 16#CEA1;
   // UNICODE_TO_GBK[9526] := 16#5DCE;
   // UNICODE_TO_GBK[9527] := 16#8E6A;
   // UNICODE_TO_GBK[9528] := 16#5DCF;
   // UNICODE_TO_GBK[9529] := 16#8E6B;
   // UNICODE_TO_GBK[9530] := 16#5DD0;
   // UNICODE_TO_GBK[9531] := 16#8E6C;
   // UNICODE_TO_GBK[9532] := 16#5DD1;
   // UNICODE_TO_GBK[9533] := 16#8E6D;
   // UNICODE_TO_GBK[9534] := 16#5DD2;
   // UNICODE_TO_GBK[9535] := 16#8E6E;
   // UNICODE_TO_GBK[9536] := 16#5DD3;
   // UNICODE_TO_GBK[9537] := 16#8E6F;
   // UNICODE_TO_GBK[9538] := 16#5DD4;
   // UNICODE_TO_GBK[9539] := 16#8E70;
   // UNICODE_TO_GBK[9540] := 16#5DD5;
   // UNICODE_TO_GBK[9541] := 16#8E71;
   // UNICODE_TO_GBK[9542] := 16#5DD6;
   // UNICODE_TO_GBK[9543] := 16#8E72;
   // UNICODE_TO_GBK[9544] := 16#5DD7;
   // UNICODE_TO_GBK[9545] := 16#8E73;
   // UNICODE_TO_GBK[9546] := 16#5DD8;
   // UNICODE_TO_GBK[9547] := 16#8E74;
   // UNICODE_TO_GBK[9548] := 16#5DD9;
   // UNICODE_TO_GBK[9549] := 16#8E75;
   // UNICODE_TO_GBK[9550] := 16#5DDA;
   // UNICODE_TO_GBK[9551] := 16#8E76;
   // UNICODE_TO_GBK[9552] := 16#5DDB;
   // UNICODE_TO_GBK[9553] := 16#E7DD;
   // UNICODE_TO_GBK[9554] := 16#5DDC;
   // UNICODE_TO_GBK[9555] := 16#8E77;
   // UNICODE_TO_GBK[9556] := 16#5DDD;
   // UNICODE_TO_GBK[9557] := 16#B4A8;
   // UNICODE_TO_GBK[9558] := 16#5DDE;
   // UNICODE_TO_GBK[9559] := 16#D6DD;
   // UNICODE_TO_GBK[9560] := 16#5DDF;
   // UNICODE_TO_GBK[9561] := 16#8E78;
   // UNICODE_TO_GBK[9562] := 16#5DE0;
   // UNICODE_TO_GBK[9563] := 16#8E79;
   // UNICODE_TO_GBK[9564] := 16#5DE1;
   // UNICODE_TO_GBK[9565] := 16#D1B2;
   // UNICODE_TO_GBK[9566] := 16#5DE2;
   // UNICODE_TO_GBK[9567] := 16#B3B2;
   // UNICODE_TO_GBK[9568] := 16#5DE3;
   // UNICODE_TO_GBK[9569] := 16#8E7A;
   // UNICODE_TO_GBK[9570] := 16#5DE4;
   // UNICODE_TO_GBK[9571] := 16#8E7B;
   // UNICODE_TO_GBK[9572] := 16#5DE5;
   // UNICODE_TO_GBK[9573] := 16#B9A4;
   // UNICODE_TO_GBK[9574] := 16#5DE6;
   // UNICODE_TO_GBK[9575] := 16#D7F3;
   // UNICODE_TO_GBK[9576] := 16#5DE7;
   // UNICODE_TO_GBK[9577] := 16#C7C9;
   // UNICODE_TO_GBK[9578] := 16#5DE8;
   // UNICODE_TO_GBK[9579] := 16#BEDE;
   // UNICODE_TO_GBK[9580] := 16#5DE9;
   // UNICODE_TO_GBK[9581] := 16#B9AE;
   // UNICODE_TO_GBK[9582] := 16#5DEA;
   // UNICODE_TO_GBK[9583] := 16#8E7C;
   // UNICODE_TO_GBK[9584] := 16#5DEB;
   // UNICODE_TO_GBK[9585] := 16#CED7;
   // UNICODE_TO_GBK[9586] := 16#5DEC;
   // UNICODE_TO_GBK[9587] := 16#8E7D;
   // UNICODE_TO_GBK[9588] := 16#5DED;
   // UNICODE_TO_GBK[9589] := 16#8E7E;
   // UNICODE_TO_GBK[9590] := 16#5DEE;
   // UNICODE_TO_GBK[9591] := 16#B2EE;
   // UNICODE_TO_GBK[9592] := 16#5DEF;
   // UNICODE_TO_GBK[9593] := 16#DBCF;
   // UNICODE_TO_GBK[9594] := 16#5DF0;
   // UNICODE_TO_GBK[9595] := 16#8E80;
   // UNICODE_TO_GBK[9596] := 16#5DF1;
   // UNICODE_TO_GBK[9597] := 16#BCBA;
   // UNICODE_TO_GBK[9598] := 16#5DF2;
   // UNICODE_TO_GBK[9599] := 16#D2D1;
   // UNICODE_TO_GBK[9600] := 16#5DF3;
   // UNICODE_TO_GBK[9601] := 16#CBC8;
   // UNICODE_TO_GBK[9602] := 16#5DF4;
   // UNICODE_TO_GBK[9603] := 16#B0CD;
   // UNICODE_TO_GBK[9604] := 16#5DF5;
   // UNICODE_TO_GBK[9605] := 16#8E81;
   // UNICODE_TO_GBK[9606] := 16#5DF6;
   // UNICODE_TO_GBK[9607] := 16#8E82;
   // UNICODE_TO_GBK[9608] := 16#5DF7;
   // UNICODE_TO_GBK[9609] := 16#CFEF;
   // UNICODE_TO_GBK[9610] := 16#5DF8;
   // UNICODE_TO_GBK[9611] := 16#8E83;
   // UNICODE_TO_GBK[9612] := 16#5DF9;
   // UNICODE_TO_GBK[9613] := 16#8E84;
   // UNICODE_TO_GBK[9614] := 16#5DFA;
   // UNICODE_TO_GBK[9615] := 16#8E85;
   // UNICODE_TO_GBK[9616] := 16#5DFB;
   // UNICODE_TO_GBK[9617] := 16#8E86;
   // UNICODE_TO_GBK[9618] := 16#5DFC;
   // UNICODE_TO_GBK[9619] := 16#8E87;
   // UNICODE_TO_GBK[9620] := 16#5DFD;
   // UNICODE_TO_GBK[9621] := 16#D9E3;
   // UNICODE_TO_GBK[9622] := 16#5DFE;
   // UNICODE_TO_GBK[9623] := 16#BDED;
   // UNICODE_TO_GBK[9624] := 16#5DFF;
   // UNICODE_TO_GBK[9625] := 16#8E88;
   // UNICODE_TO_GBK[9626] := 16#5E00;
   // UNICODE_TO_GBK[9627] := 16#8E89;
   // UNICODE_TO_GBK[9628] := 16#5E01;
   // UNICODE_TO_GBK[9629] := 16#B1D2;
   // UNICODE_TO_GBK[9630] := 16#5E02;
   // UNICODE_TO_GBK[9631] := 16#CAD0;
   // UNICODE_TO_GBK[9632] := 16#5E03;
   // UNICODE_TO_GBK[9633] := 16#B2BC;
   // UNICODE_TO_GBK[9634] := 16#5E04;
   // UNICODE_TO_GBK[9635] := 16#8E8A;
   // UNICODE_TO_GBK[9636] := 16#5E05;
   // UNICODE_TO_GBK[9637] := 16#CBA7;
   // UNICODE_TO_GBK[9638] := 16#5E06;
   // UNICODE_TO_GBK[9639] := 16#B7AB;
   // UNICODE_TO_GBK[9640] := 16#5E07;
   // UNICODE_TO_GBK[9641] := 16#8E8B;
   // UNICODE_TO_GBK[9642] := 16#5E08;
   // UNICODE_TO_GBK[9643] := 16#CAA6;
   // UNICODE_TO_GBK[9644] := 16#5E09;
   // UNICODE_TO_GBK[9645] := 16#8E8C;
   // UNICODE_TO_GBK[9646] := 16#5E0A;
   // UNICODE_TO_GBK[9647] := 16#8E8D;
   // UNICODE_TO_GBK[9648] := 16#5E0B;
   // UNICODE_TO_GBK[9649] := 16#8E8E;
   // UNICODE_TO_GBK[9650] := 16#5E0C;
   // UNICODE_TO_GBK[9651] := 16#CFA3;
   // UNICODE_TO_GBK[9652] := 16#5E0D;
   // UNICODE_TO_GBK[9653] := 16#8E8F;
   // UNICODE_TO_GBK[9654] := 16#5E0E;
   // UNICODE_TO_GBK[9655] := 16#8E90;
   // UNICODE_TO_GBK[9656] := 16#5E0F;
   // UNICODE_TO_GBK[9657] := 16#E0F8;
   // UNICODE_TO_GBK[9658] := 16#5E10;
   // UNICODE_TO_GBK[9659] := 16#D5CA;
   // UNICODE_TO_GBK[9660] := 16#5E11;
   // UNICODE_TO_GBK[9661] := 16#E0FB;
   // UNICODE_TO_GBK[9662] := 16#5E12;
   // UNICODE_TO_GBK[9663] := 16#8E91;
   // UNICODE_TO_GBK[9664] := 16#5E13;
   // UNICODE_TO_GBK[9665] := 16#8E92;
   // UNICODE_TO_GBK[9666] := 16#5E14;
   // UNICODE_TO_GBK[9667] := 16#E0FA;
   // UNICODE_TO_GBK[9668] := 16#5E15;
   // UNICODE_TO_GBK[9669] := 16#C5C1;
   // UNICODE_TO_GBK[9670] := 16#5E16;
   // UNICODE_TO_GBK[9671] := 16#CCFB;
   // UNICODE_TO_GBK[9672] := 16#5E17;
   // UNICODE_TO_GBK[9673] := 16#8E93;
   // UNICODE_TO_GBK[9674] := 16#5E18;
   // UNICODE_TO_GBK[9675] := 16#C1B1;
   // UNICODE_TO_GBK[9676] := 16#5E19;
   // UNICODE_TO_GBK[9677] := 16#E0F9;
   // UNICODE_TO_GBK[9678] := 16#5E1A;
   // UNICODE_TO_GBK[9679] := 16#D6E3;
   // UNICODE_TO_GBK[9680] := 16#5E1B;
   // UNICODE_TO_GBK[9681] := 16#B2AF;
   // UNICODE_TO_GBK[9682] := 16#5E1C;
   // UNICODE_TO_GBK[9683] := 16#D6C4;
   // UNICODE_TO_GBK[9684] := 16#5E1D;
   // UNICODE_TO_GBK[9685] := 16#B5DB;
   // UNICODE_TO_GBK[9686] := 16#5E1E;
   // UNICODE_TO_GBK[9687] := 16#8E94;
   // UNICODE_TO_GBK[9688] := 16#5E1F;
   // UNICODE_TO_GBK[9689] := 16#8E95;
   // UNICODE_TO_GBK[9690] := 16#5E20;
   // UNICODE_TO_GBK[9691] := 16#8E96;
   // UNICODE_TO_GBK[9692] := 16#5E21;
   // UNICODE_TO_GBK[9693] := 16#8E97;
   // UNICODE_TO_GBK[9694] := 16#5E22;
   // UNICODE_TO_GBK[9695] := 16#8E98;
   // UNICODE_TO_GBK[9696] := 16#5E23;
   // UNICODE_TO_GBK[9697] := 16#8E99;
   // UNICODE_TO_GBK[9698] := 16#5E24;
   // UNICODE_TO_GBK[9699] := 16#8E9A;
   // UNICODE_TO_GBK[9700] := 16#5E25;
   // UNICODE_TO_GBK[9701] := 16#8E9B;
   // UNICODE_TO_GBK[9702] := 16#5E26;
   // UNICODE_TO_GBK[9703] := 16#B4F8;
   // UNICODE_TO_GBK[9704] := 16#5E27;
   // UNICODE_TO_GBK[9705] := 16#D6A1;
   // UNICODE_TO_GBK[9706] := 16#5E28;
   // UNICODE_TO_GBK[9707] := 16#8E9C;
   // UNICODE_TO_GBK[9708] := 16#5E29;
   // UNICODE_TO_GBK[9709] := 16#8E9D;
   // UNICODE_TO_GBK[9710] := 16#5E2A;
   // UNICODE_TO_GBK[9711] := 16#8E9E;
   // UNICODE_TO_GBK[9712] := 16#5E2B;
   // UNICODE_TO_GBK[9713] := 16#8E9F;
   // UNICODE_TO_GBK[9714] := 16#5E2C;
   // UNICODE_TO_GBK[9715] := 16#8EA0;
   // UNICODE_TO_GBK[9716] := 16#5E2D;
   // UNICODE_TO_GBK[9717] := 16#CFAF;
   // UNICODE_TO_GBK[9718] := 16#5E2E;
   // UNICODE_TO_GBK[9719] := 16#B0EF;
   // UNICODE_TO_GBK[9720] := 16#5E2F;
   // UNICODE_TO_GBK[9721] := 16#8EA1;
   // UNICODE_TO_GBK[9722] := 16#5E30;
   // UNICODE_TO_GBK[9723] := 16#8EA2;
   // UNICODE_TO_GBK[9724] := 16#5E31;
   // UNICODE_TO_GBK[9725] := 16#E0FC;
   // UNICODE_TO_GBK[9726] := 16#5E32;
   // UNICODE_TO_GBK[9727] := 16#8EA3;
   // UNICODE_TO_GBK[9728] := 16#5E33;
   // UNICODE_TO_GBK[9729] := 16#8EA4;
   // UNICODE_TO_GBK[9730] := 16#5E34;
   // UNICODE_TO_GBK[9731] := 16#8EA5;
   // UNICODE_TO_GBK[9732] := 16#5E35;
   // UNICODE_TO_GBK[9733] := 16#8EA6;
   // UNICODE_TO_GBK[9734] := 16#5E36;
   // UNICODE_TO_GBK[9735] := 16#8EA7;
   // UNICODE_TO_GBK[9736] := 16#5E37;
   // UNICODE_TO_GBK[9737] := 16#E1A1;
   // UNICODE_TO_GBK[9738] := 16#5E38;
   // UNICODE_TO_GBK[9739] := 16#B3A3;
   // UNICODE_TO_GBK[9740] := 16#5E39;
   // UNICODE_TO_GBK[9741] := 16#8EA8;
   // UNICODE_TO_GBK[9742] := 16#5E3A;
   // UNICODE_TO_GBK[9743] := 16#8EA9;
   // UNICODE_TO_GBK[9744] := 16#5E3B;
   // UNICODE_TO_GBK[9745] := 16#E0FD;
   // UNICODE_TO_GBK[9746] := 16#5E3C;
   // UNICODE_TO_GBK[9747] := 16#E0FE;
   // UNICODE_TO_GBK[9748] := 16#5E3D;
   // UNICODE_TO_GBK[9749] := 16#C3B1;
   // UNICODE_TO_GBK[9750] := 16#5E3E;
   // UNICODE_TO_GBK[9751] := 16#8EAA;
   // UNICODE_TO_GBK[9752] := 16#5E3F;
   // UNICODE_TO_GBK[9753] := 16#8EAB;
   // UNICODE_TO_GBK[9754] := 16#5E40;
   // UNICODE_TO_GBK[9755] := 16#8EAC;
   // UNICODE_TO_GBK[9756] := 16#5E41;
   // UNICODE_TO_GBK[9757] := 16#8EAD;
   // UNICODE_TO_GBK[9758] := 16#5E42;
   // UNICODE_TO_GBK[9759] := 16#C3DD;
   // UNICODE_TO_GBK[9760] := 16#5E43;
   // UNICODE_TO_GBK[9761] := 16#8EAE;
   // UNICODE_TO_GBK[9762] := 16#5E44;
   // UNICODE_TO_GBK[9763] := 16#E1A2;
   // UNICODE_TO_GBK[9764] := 16#5E45;
   // UNICODE_TO_GBK[9765] := 16#B7F9;
   // UNICODE_TO_GBK[9766] := 16#5E46;
   // UNICODE_TO_GBK[9767] := 16#8EAF;
   // UNICODE_TO_GBK[9768] := 16#5E47;
   // UNICODE_TO_GBK[9769] := 16#8EB0;
   // UNICODE_TO_GBK[9770] := 16#5E48;
   // UNICODE_TO_GBK[9771] := 16#8EB1;
   // UNICODE_TO_GBK[9772] := 16#5E49;
   // UNICODE_TO_GBK[9773] := 16#8EB2;
   // UNICODE_TO_GBK[9774] := 16#5E4A;
   // UNICODE_TO_GBK[9775] := 16#8EB3;
   // UNICODE_TO_GBK[9776] := 16#5E4B;
   // UNICODE_TO_GBK[9777] := 16#8EB4;
   // UNICODE_TO_GBK[9778] := 16#5E4C;
   // UNICODE_TO_GBK[9779] := 16#BBCF;
   // UNICODE_TO_GBK[9780] := 16#5E4D;
   // UNICODE_TO_GBK[9781] := 16#8EB5;
   // UNICODE_TO_GBK[9782] := 16#5E4E;
   // UNICODE_TO_GBK[9783] := 16#8EB6;
   // UNICODE_TO_GBK[9784] := 16#5E4F;
   // UNICODE_TO_GBK[9785] := 16#8EB7;
   // UNICODE_TO_GBK[9786] := 16#5E50;
   // UNICODE_TO_GBK[9787] := 16#8EB8;
   // UNICODE_TO_GBK[9788] := 16#5E51;
   // UNICODE_TO_GBK[9789] := 16#8EB9;
   // UNICODE_TO_GBK[9790] := 16#5E52;
   // UNICODE_TO_GBK[9791] := 16#8EBA;
   // UNICODE_TO_GBK[9792] := 16#5E53;
   // UNICODE_TO_GBK[9793] := 16#8EBB;
   // UNICODE_TO_GBK[9794] := 16#5E54;
   // UNICODE_TO_GBK[9795] := 16#E1A3;
   // UNICODE_TO_GBK[9796] := 16#5E55;
   // UNICODE_TO_GBK[9797] := 16#C4BB;
   // UNICODE_TO_GBK[9798] := 16#5E56;
   // UNICODE_TO_GBK[9799] := 16#8EBC;
   // UNICODE_TO_GBK[9800] := 16#5E57;
   // UNICODE_TO_GBK[9801] := 16#8EBD;
   // UNICODE_TO_GBK[9802] := 16#5E58;
   // UNICODE_TO_GBK[9803] := 16#8EBE;
   // UNICODE_TO_GBK[9804] := 16#5E59;
   // UNICODE_TO_GBK[9805] := 16#8EBF;
   // UNICODE_TO_GBK[9806] := 16#5E5A;
   // UNICODE_TO_GBK[9807] := 16#8EC0;
   // UNICODE_TO_GBK[9808] := 16#5E5B;
   // UNICODE_TO_GBK[9809] := 16#E1A4;
   // UNICODE_TO_GBK[9810] := 16#5E5C;
   // UNICODE_TO_GBK[9811] := 16#8EC1;
   // UNICODE_TO_GBK[9812] := 16#5E5D;
   // UNICODE_TO_GBK[9813] := 16#8EC2;
   // UNICODE_TO_GBK[9814] := 16#5E5E;
   // UNICODE_TO_GBK[9815] := 16#E1A5;
   // UNICODE_TO_GBK[9816] := 16#5E5F;
   // UNICODE_TO_GBK[9817] := 16#8EC3;
   // UNICODE_TO_GBK[9818] := 16#5E60;
   // UNICODE_TO_GBK[9819] := 16#8EC4;
   // UNICODE_TO_GBK[9820] := 16#5E61;
   // UNICODE_TO_GBK[9821] := 16#E1A6;
